# B&R Automation Studio project OpcUaSample410_BrbLibUa103 (part 15)

#### autoGeneratedFile.c - Auto generated code - list of all test sets in the program
```c
/*
B+R UnitTest: This is generated code.
Do not edit! Do not move!
Description: UnitTest Testprogramm infrastructure (List of TestSets).
LastUpdated: 2023-04-20 12:30:26Z
By B+R UnitTest Helper Version: 2.0.1.59
*/
#include "UnitTest.h"

UNITTEST_TESTSET_DECLARATION  Set_BrbUaClearVariantValue;
UNITTEST_TESTSET_DECLARATION  Set_BrbUaConvVariantValueFromString;
UNITTEST_TESTSET_DECLARATION  Set_BrbUaConvVariantValueToString;
UNITTEST_TESTSET_DECLARATION  Set_BrbUaAddVariantValueSubName;

UNITTEST_TESTSET_FIXTURES(utTestSets)
{
	new_TestSet(Set_BrbUaClearVariantValue),
	new_TestSet(Set_BrbUaConvVariantValueFromString),
	new_TestSet(Set_BrbUaConvVariantValueToString),
	new_TestSet(Set_BrbUaAddVariantValueSubName),
};
UNTITTEST_TESTSET_HANDLER();
```

#### Set_BrbUaClearVariantValue.c - Test set
```c
#include <bur/plctypes.h>

#ifdef _DEFAULT_INCLUDES
#include <AsDefault.h>
#endif

#include "UnitTest.h"
#include "BrbAsserts.h"
#include <string.h>

// NOLINTBEGIN(readability-*, bugprone-easily-swappable-parameters, bugprone-branch-clone, clang-diagnostic-invalid-utf8, clang-diagnostic-invalid-source-encoding, clang-diagnostic-pointer-arith, clang-diagnostic-strict-prototypes, clang-diagnostic-bad-function-cast, clang-analyzer-security.insecureAPI.*, hicpp-uppercase-literal-suffix, cppcoreguidelines-*, performance-*)
_TEST BrbUaClearVariantValue_NulPtr(void)
{
	dwordOut = BrbUaClearVariantValue(0);
	TEST_ASSERT_EQUAL_INT(0x80460000, dwordOut); // = Bad_StructureMissing

	// Finished
	TEST_DONE;
}

_TEST BrbUaClearVariantValue_Clear(void)
{
	memset(&variantIn0, 1, sizeof(variantIn0));
	variantIn0.VariantType = UAVariantType_Byte;
	dwordOut = BrbUaClearVariantValue(&variantIn0);
	TEST_ASSERT_EQUAL_INT(0x00000000, dwordOut); // = Good
	BRB_ASSERT_EQUAL_DINT(UAVariantType_Byte, (DINT)variantIn0.VariantType);

	// Finished
	TEST_DONE;
}

// NOLINTEND(readability-*, bugprone-easily-swappable-parameters, bugprone-branch-clone, clang-diagnostic-invalid-utf8, clang-diagnostic-invalid-source-encoding, clang-diagnostic-pointer-arith, clang-diagnostic-strict-prototypes, clang-diagnostic-bad-function-cast, clang-analyzer-security.insecureAPI.*, hicpp-uppercase-literal-suffix, cppcoreguidelines-*, performance-*)

/*
B+R UnitTest: This is generated code.
Do not edit! Do not move!
Description: UnitTest Testprogramm infrastructure (TestSet).
LastUpdated: 2023-04-20 10:55:13Z
By B+R UnitTest Helper Version: 2.0.1.59
*/
UNITTEST_FIXTURES(fixtures)
{
	new_TestFixture("BrbUaClearVariantValue_NulPtr", BrbUaClearVariantValue_NulPtr),
	new_TestFixture("BrbUaClearVariantValue_Clear", BrbUaClearVariantValue_Clear),
};

UNITTEST_CALLER_COMPLETE_EXPLICIT(Set_BrbUaClearVariantValue, "Set_BrbUaClearVariantValue", 0, 0, fixtures, 0, 0, 0);
```

#### Set_BrbUaConvVariantValueFromString.c - Test set
```c
#include <bur/plctypes.h>

#ifdef _DEFAULT_INCLUDES
#include <AsDefault.h>
#endif

#include "UnitTest.h"
#include "BrbAsserts.h"
#include <string.h>

// NOLINTBEGIN(readability-*, bugprone-easily-swappable-parameters, bugprone-branch-clone, clang-diagnostic-invalid-utf8, clang-diagnostic-invalid-source-encoding, clang-diagnostic-pointer-arith, clang-diagnostic-strict-prototypes, clang-diagnostic-bad-function-cast, clang-analyzer-security.insecureAPI.*, hicpp-uppercase-literal-suffix, cppcoreguidelines-*, performance-*)
_TEST BrbUaConvVariantValueFromString_NulPtr(void)
{
	dwordOut = BrbUaConvVariantValueFromString(0, stringIn0);
	TEST_ASSERT_EQUAL_INT(0x80460000, dwordOut); // = Bad_StructureMissing

	dwordOut = BrbUaConvVariantValueFromString(&variantIn0, 0);
	TEST_ASSERT_EQUAL_INT(0x80460000, dwordOut); // = Bad_StructureMissing

	// Finished
	TEST_DONE;
}

_TEST BrbUaConvVariantValueFromString_Boolean(void)
{
	memset(&variantIn0, 0, sizeof(variantIn0));
	variantIn0.VariantType = UAVariantType_Boolean;
	strcpy(stringIn0, "xxx");
	dwordOut = BrbUaConvVariantValueFromString(&variantIn0, stringIn0);
	TEST_ASSERT_EQUAL_INT(0x00000000, dwordOut); // = Good
	BRB_ASSERT_EQUAL_DINT(UAVariantType_Boolean, (DINT)variantIn0.VariantType);
	BRB_ASSERT_EQUAL_BOOL(0, variantIn0.Boolean);

	memset(&variantIn0, 0, sizeof(variantIn0));
	variantIn0.VariantType = UAVariantType_Boolean;
	strcpy(stringIn0, "0");
	dwordOut = BrbUaConvVariantValueFromString(&variantIn0, stringIn0);
	TEST_ASSERT_EQUAL_INT(0x00000000, dwordOut); // = Good
	BRB_ASSERT_EQUAL_DINT(UAVariantType_Boolean, (DINT)variantIn0.VariantType);
	BRB_ASSERT_EQUAL_BOOL(0, variantIn0.Boolean);

	memset(&variantIn0, 0, sizeof(variantIn0));
	variantIn0.VariantType = UAVariantType_Boolean;
	strcpy(stringIn0, "False");
	dwordOut = BrbUaConvVariantValueFromString(&variantIn0, stringIn0);
	TEST_ASSERT_EQUAL_INT(0x00000000, dwordOut); // = Good
	BRB_ASSERT_EQUAL_DINT(UAVariantType_Boolean, (DINT)variantIn0.VariantType);
	BRB_ASSERT_EQUAL_BOOL(0, variantIn0.Boolean);

	memset(&variantIn0, 0, sizeof(variantIn0));
	variantIn0.VariantType = UAVariantType_Boolean;
	strcpy(stringIn0, "false");
	dwordOut = BrbUaConvVariantValueFromString(&variantIn0, stringIn0);
	TEST_ASSERT_EQUAL_INT(0x00000000, dwordOut); // = Good
	BRB_ASSERT_EQUAL_DINT(UAVariantType_Boolean, (DINT)variantIn0.VariantType);
	BRB_ASSERT_EQUAL_BOOL(0, variantIn0.Boolean);

	memset(&variantIn0, 0, sizeof(variantIn0));
	variantIn0.VariantType = UAVariantType_Boolean;
	strcpy(stringIn0, "1");
	dwordOut = BrbUaConvVariantValueFromString(&variantIn0, stringIn0);
	TEST_ASSERT_EQUAL_INT(0x00000000, dwordOut); // = Good
	BRB_ASSERT_EQUAL_DINT(UAVariantType_Boolean, (DINT)variantIn0.VariantType);
	BRB_ASSERT_EQUAL_BOOL(1, variantIn0.Boolean);

	memset(&variantIn0, 0, sizeof(variantIn0));
	variantIn0.VariantType = UAVariantType_Boolean;
	strcpy(stringIn0, "True");
	dwordOut = BrbUaConvVariantValueFromString(&variantIn0, stringIn0);
	TEST_ASSERT_EQUAL_INT(0x00000000, dwordOut); // = Good
	BRB_ASSERT_EQUAL_DINT(UAVariantType_Boolean, (DINT)variantIn0.VariantType);
	BRB_ASSERT_EQUAL_BOOL(1, variantIn0.Boolean);

	memset(&variantIn0, 0, sizeof(variantIn0));
	variantIn0.VariantType = UAVariantType_Boolean;
	strcpy(stringIn0, "true");
	dwordOut = BrbUaConvVariantValueFromString(&variantIn0, stringIn0);
	TEST_ASSERT_EQUAL_INT(0x00000000, dwordOut); // = Good
	BRB_ASSERT_EQUAL_DINT(UAVariantType_Boolean, (DINT)variantIn0.VariantType);
	BRB_ASSERT_EQUAL_BOOL(1, variantIn0.Boolean);

	// Finished
	TEST_DONE;
}

_TEST BrbUaConvVariantValueFromString_SByte(void)
{
	memset(&variantIn0, 0, sizeof(variantIn0));
	variantIn0.VariantType = UAVariantType_SByte;
	strcpy(stringIn0, "-128");
	dwordOut = BrbUaConvVariantValueFromString(&variantIn0, stringIn0);
	TEST_ASSERT_EQUAL_INT(0x00000000, dwordOut); // = Good
	BRB_ASSERT_EQUAL_DINT(UAVariantType_SByte, (DINT)variantIn0.VariantType);
	BRB_ASSERT_EQUAL_DINT(-128, (DINT)variantIn0.SByte);

	// Finished
	TEST_DONE;
}

_TEST BrbUaConvVariantValueFromString_Byte(void)
{
	memset(&variantIn0, 0, sizeof(variantIn0));
	variantIn0.VariantType = UAVariantType_Byte;
	strcpy(stringIn0, "127");
	dwordOut = BrbUaConvVariantValueFromString(&variantIn0, stringIn0);
	TEST_ASSERT_EQUAL_INT(0x00000000, dwordOut); // = Good
	BRB_ASSERT_EQUAL_DINT(UAVariantType_Byte, (DINT)variantIn0.VariantType);
	BRB_ASSERT_EQUAL_UDINT(127, (UDINT)variantIn0.Byte);

	// Finished
	TEST_DONE;
}

_TEST BrbUaConvVariantValueFromString_Int16(void)
{
	memset(&variantIn0, 0, sizeof(variantIn0));
	variantIn0.VariantType = UAVariantType_Int16;
	strcpy(stringIn0, "-32768");
	dwordOut = BrbUaConvVariantValueFromString(&variantIn0, stringIn0);
	TEST_ASSERT_EQUAL_INT(0x00000000, dwordOut); // = Good
	BRB_ASSERT_EQUAL_DINT(UAVariantType_Int16, (DINT)variantIn0.VariantType);
	BRB_ASSERT_EQUAL_DINT(-32768, (DINT)variantIn0.Int16);

	// Finished
	TEST_DONE;
}

_TEST BrbUaConvVariantValueFromString_Uint16(void)
{
	memset(&variantIn0, 0, sizeof(variantIn0));
	variantIn0.VariantType = UAVariantType_UInt16;
	strcpy(stringIn0, "65535");
	dwordOut = BrbUaConvVariantValueFromString(&variantIn0, stringIn0);
	TEST_ASSERT_EQUAL_INT(0x00000000, dwordOut); // = Good
	BRB_ASSERT_EQUAL_DINT(UAVariantType_UInt16, (DINT)variantIn0.VariantType);
	BRB_ASSERT_EQUAL_UDINT(65535, (UDINT)variantIn0.UInt16);

	// Finished
	TEST_DONE;
}

_TEST BrbUaConvVariantValueFromString_Int32(void)
{
	memset(&variantIn0, 0, sizeof(variantIn0));
	variantIn0.VariantType = UAVariantType_Int32;
	strcpy(stringIn0, "-2147483648");
	dwordOut = BrbUaConvVariantValueFromString(&variantIn0, stringIn0);
	TEST_ASSERT_EQUAL_INT(0x00000000, dwordOut); // = Good
	BRB_ASSERT_EQUAL_DINT(UAVariantType_Int32, (DINT)variantIn0.VariantType);
	BRB_ASSERT_EQUAL_DINT(-2147483648, (DINT)variantIn0.Int32);

	// Finished
	TEST_DONE;
}

_TEST BrbUaConvVariantValueFromString_Uint32(void)
{
	memset(&variantIn0, 0, sizeof(variantIn0));
	variantIn0.VariantType = UAVariantType_UInt32;
	strcpy(stringIn0, "4294967295");
	dwordOut = BrbUaConvVariantValueFromString(&variantIn0, stringIn0);
	TEST_ASSERT_EQUAL_INT(0x00000000, dwordOut); // = Good
	BRB_ASSERT_EQUAL_DINT(UAVariantType_UInt32, (DINT)variantIn0.VariantType);
	BRB_ASSERT_EQUAL_UDINT(4294967295, variantIn0.UInt32);

	// Finished
	TEST_DONE;
}

_TEST BrbUaConvVariantValueFromString_Int64(void)
{
	memset(&variantIn0, 0, sizeof(variantIn0));
	variantIn0.VariantType = UAVariantType_Int64;
	strcpy(stringIn0, "-2147483648");
	dwordOut = BrbUaConvVariantValueFromString(&variantIn0, stringIn0);
	TEST_ASSERT_EQUAL_INT(0x803D0000, dwordOut); // = Bad_NotSupported
	BRB_ASSERT_EQUAL_DINT(UAVariantType_Int64, (DINT)variantIn0.VariantType);

	// Finished
	TEST_DONE;
}

_TEST BrbUaConvVariantValueFromString_Uint64(void)
{
	memset(&variantIn0, 0, sizeof(variantIn0));
	variantIn0.VariantType = UAVariantType_UInt64;
	strcpy(stringIn0, "4294967295");
	dwordOut = BrbUaConvVariantValueFromString(&variantIn0, stringIn0);
	TEST_ASSERT_EQUAL_INT(0x803D0000, dwordOut); // = Bad_NotSupported
	BRB_ASSERT_EQUAL_DINT(UAVariantType_UInt64, (DINT)variantIn0.VariantType);

	// Finished
	TEST_DONE;
}

_TEST BrbUaConvVariantValueFromString_Float(void)
{
	memset(&variantIn0, 0, sizeof(variantIn0));
	variantIn0.VariantType = UAVariantType_Float;
	strcpy(stringIn0, "-1.23");
	dwordOut = BrbUaConvVariantValueFromString(&variantIn0, stringIn0);
	TEST_ASSERT_EQUAL_INT(0x00000000, dwordOut); // = Good
	BRB_ASSERT_EQUAL_DINT(UAVariantType_Float, (DINT)variantIn0.VariantType);
	TEST_ASSERT_EQUAL_REAL(-1.23, variantIn0.Float);

	// Finished
	TEST_DONE;
}

_TEST BrbUaConvVariantValueFromString_Double(void)
{
	memset(&variantIn0, 0, sizeof(variantIn0));
	variantIn0.VariantType = UAVariantType_Double;
	strcpy(stringIn0, "-2.34");
	dwordOut = BrbUaConvVariantValueFromString(&variantIn0, stringIn0);
	TEST_ASSERT_EQUAL_INT(0x00000000, dwordOut); // = Good
	BRB_ASSERT_EQUAL_DINT(UAVariantType_Double, (DINT)variantIn0.VariantType);
	TEST_ASSERT_EQUAL_LREAL((LREAL)-2.3399999141693115, variantIn0.Double);

	// Finished
	TEST_DONE;
}

_TEST BrbUaConvVariantValueFromString_String(void)
{
	memset(&variantIn0, 0, sizeof(variantIn0));
	variantIn0.VariantType = UAVariantType_String;
	strcpy(stringIn0, "Hallo");
	dwordOut = BrbUaConvVariantValueFromString(&variantIn0, stringIn0);
	TEST_ASSERT_EQUAL_INT(0x00000000, dwordOut); // = Good
	BRB_ASSERT_EQUAL_DINT(UAVariantType_String, (DINT)variantIn0.VariantType);
	TEST_ASSERT_EQUAL_STRING("Hallo", variantIn0.String);

	// Finished
	TEST_DONE;
}

_TEST BrbUaConvVariantValueFromString_DateTime(void)
{
	memset(&variantIn0, 0, sizeof(variantIn0));
	variantIn0.VariantType = UAVariantType_DateTime;
	strcpy(stringIn0, "2106.02.07 06:28:15:000:000");
	dwordOut = BrbUaConvVariantValueFromString(&variantIn0, stringIn0);
	TEST_ASSERT_EQUAL_INT(0x00000000, dwordOut); // = Good
	BRB_ASSERT_EQUAL_DINT(UAVariantType_DateTime, (DINT)variantIn0.VariantType);
	BRB_ASSERT_EQUAL_UDINT(4294967295, (UDINT)variantIn0.DateTime);

	// Finished
	TEST_DONE;
}

_TEST BrbUaConvVariantValueFromString_Guid(void)
{
	memset(&variantIn0, 0, sizeof(variantIn0));
	variantIn0.VariantType = UAVariantType_Guid;
	strcpy(stringIn0, "12345678-1234-5678-9ABC-123456789ABC");
	dwordOut = BrbUaConvVariantValueFromString(&variantIn0, stringIn0);
	TEST_ASSERT_EQUAL_INT(0x00000000, dwordOut); // = Good
	BRB_ASSERT_EQUAL_DINT(UAVariantType_Guid, (DINT)variantIn0.VariantType);
	TEST_ASSERT_EQUAL_STRING("12345678-1234-5678-9ABC-123456789ABC", variantIn0.String);

	// Finished
	TEST_DONE;
}

_TEST BrbUaConvVariantValueFromString_ByteString(void)
{
	memset(&variantIn0, 0, sizeof(variantIn0));
	variantIn0.VariantType = UAVariantType_ByteString;
	strcpy(stringIn0, "123456789ABC");
	dwordOut = BrbUaConvVariantValueFromString(&variantIn0, stringIn0);
	TEST_ASSERT_EQUAL_INT(0x803D0000, dwordOut); // = Bad_NotSupported
	BRB_ASSERT_EQUAL_DINT(UAVariantType_ByteString, (DINT)variantIn0.VariantType);

	// Finished
	TEST_DONE;
}

_TEST BrbUaConvVariantValueFromString_XmlElement(void)
{
	memset(&variantIn0, 0, sizeof(variantIn0));
	variantIn0.VariantType = UAVariantType_XmlElement;
	strcpy(stringIn0, "<Hallo >");
	dwordOut = BrbUaConvVariantValueFromString(&variantIn0, stringIn0);
	TEST_ASSERT_EQUAL_INT(0x803D0000, dwordOut); // = Bad_NotSupported
	BRB_ASSERT_EQUAL_DINT(UAVariantType_XmlElement, (DINT)variantIn0.VariantType);

	// Finished
	TEST_DONE;
}

_TEST BrbUaConvVariantValueFromString_NodeId(void)
{
	memset(&variantIn0, 0, sizeof(variantIn0));
	variantIn0.VariantType = UAVariantType_NodeId;
	strcpy(stringIn0, "ns=34");
	dwordOut = BrbUaConvVariantValueFromString(&variantIn0, stringIn0);
	TEST_ASSERT_EQUAL_INT(0x80330000 , dwordOut); // = Bad_NodeIdInvalid
	BRB_ASSERT_EQUAL_DINT(UAVariantType_NodeId, (DINT)variantIn0.VariantType);
	BRB_ASSERT_EQUAL_UDINT(34, (UDINT)variantIn0.NodeId.NamespaceIndex);
	//BRB_ASSERT_EQUAL_DINT(UAIdentifierType_Numeric, variantIn0.NodeId.IdentifierType);
	TEST_ASSERT_EQUAL_STRING("", variantIn0.NodeId.Identifier);

	memset(&variantIn0, 0, sizeof(variantIn0));
	variantIn0.VariantType = UAVariantType_NodeId;
	strcpy(stringIn0, "ns=56;");
	dwordOut = BrbUaConvVariantValueFromString(&variantIn0, stringIn0);
	TEST_ASSERT_EQUAL_INT(0x80330000 , dwordOut); // = Bad_NodeIdInvalid
	BRB_ASSERT_EQUAL_DINT(UAVariantType_NodeId, (DINT)variantIn0.VariantType);
	BRB_ASSERT_EQUAL_UDINT(56, (UDINT)variantIn0.NodeId.NamespaceIndex);
	//BRB_ASSERT_EQUAL_DINT(UAIdentifierType_Numeric, variantIn0.NodeId.IdentifierType);
	TEST_ASSERT_EQUAL_STRING("", variantIn0.NodeId.Identifier);

	memset(&variantIn0, 0, sizeof(variantIn0));
	variantIn0.VariantType = UAVariantType_NodeId;
	strcpy(stringIn0, "ns=123;v=Hallo");
	dwordOut = BrbUaConvVariantValueFromString(&variantIn0, stringIn0);
	TEST_ASSERT_EQUAL_INT(0x80330000 , dwordOut); // = Bad_NodeIdInvalid
	BRB_ASSERT_EQUAL_DINT(UAVariantType_NodeId, (DINT)variantIn0.VariantType);
	BRB_ASSERT_EQUAL_UDINT(123, (UDINT)variantIn0.NodeId.NamespaceIndex);
	//BRB_ASSERT_EQUAL_DINT(UAIdentifierType_Numeric, variantIn0.NodeId.IdentifierType);
	TEST_ASSERT_EQUAL_STRING("", variantIn0.NodeId.Identifier);

	memset(&variantIn0, 0, sizeof(variantIn0));
	variantIn0.VariantType = UAVariantType_NodeId;
	strcpy(stringIn0, "i=1234");
	dwordOut = BrbUaConvVariantValueFromString(&variantIn0, stringIn0);
	TEST_ASSERT_EQUAL_INT(0x00000000, dwordOut); // = Good
	BRB_ASSERT_EQUAL_DINT(UAVariantType_NodeId, (DINT)variantIn0.VariantType);
	BRB_ASSERT_EQUAL_UDINT(0, (UDINT)variantIn0.NodeId.NamespaceIndex);
	BRB_ASSERT_EQUAL_DINT(UAIdentifierType_Numeric, (DINT)variantIn0.NodeId.IdentifierType);
	TEST_ASSERT_EQUAL_STRING("1234", variantIn0.NodeId.Identifier);

	memset(&variantIn0, 0, sizeof(variantIn0));
	variantIn0.VariantType = UAVariantType_NodeId;
	strcpy(stringIn0, "ns=21;i=2345");
	dwordOut = BrbUaConvVariantValueFromString(&variantIn0, stringIn0);
	TEST_ASSERT_EQUAL_INT(0x00000000, dwordOut); // = Good
	BRB_ASSERT_EQUAL_DINT(UAVariantType_NodeId, (DINT)variantIn0.VariantType);
	BRB_ASSERT_EQUAL_UDINT(21, (UDINT)variantIn0.NodeId.NamespaceIndex);
	BRB_ASSERT_EQUAL_DINT(UAIdentifierType_Numeric, (DINT)variantIn0.NodeId.IdentifierType);
	TEST_ASSERT_EQUAL_STRING("2345", variantIn0.NodeId.Identifier);

	memset(&variantIn0, 0, sizeof(variantIn0));
	variantIn0.VariantType = UAVariantType_NodeId;
	strcpy(stringIn0, "s=Hallo");
	dwordOut = BrbUaConvVariantValueFromString(&variantIn0, stringIn0);
	TEST_ASSERT_EQUAL_INT(0x00000000, dwordOut); // = Good
	BRB_ASSERT_EQUAL_DINT(UAVariantType_NodeId, (DINT)variantIn0.VariantType);
	BRB_ASSERT_EQUAL_UDINT(0, (UDINT)variantIn0.NodeId.NamespaceIndex);
	BRB_ASSERT_EQUAL_DINT(UAIdentifierType_String, (DINT)variantIn0.NodeId.IdentifierType);
	TEST_ASSERT_EQUAL_STRING("Hallo", variantIn0.NodeId.Identifier);

	memset(&variantIn0, 0, sizeof(variantIn0));
	variantIn0.VariantType = UAVariantType_NodeId;
	strcpy(stringIn0, "ns=22;s=Hello");
	dwordOut = BrbUaConvVariantValueFromString(&variantIn0, stringIn0);
	TEST_ASSERT_EQUAL_INT(0x00000000, dwordOut); // = Good
	BRB_ASSERT_EQUAL_DINT(UAVariantType_NodeId, (DINT)variantIn0.VariantType);
	BRB_ASSERT_EQUAL_UDINT(22, (UDINT)variantIn0.NodeId.NamespaceIndex);
	BRB_ASSERT_EQUAL_DINT(UAIdentifierType_String, (DINT)variantIn0.NodeId.IdentifierType);
	TEST_ASSERT_EQUAL_STRING("Hello", variantIn0.NodeId.Identifier);

	memset(&variantIn0, 0, sizeof(variantIn0));
	variantIn0.VariantType = UAVariantType_NodeId;
	strcpy(stringIn0, "g=7fdf25f9-7815-e783-488b-a4247f55b88e");
	dwordOut = BrbUaConvVariantValueFromString(&variantIn0, stringIn0);
	TEST_ASSERT_EQUAL_INT(0x00000000, dwordOut); // = Good
	BRB_ASSERT_EQUAL_DINT(UAVariantType_NodeId, (DINT)variantIn0.VariantType);
	BRB_ASSERT_EQUAL_UDINT(0, (UDINT)variantIn0.NodeId.NamespaceIndex);
	BRB_ASSERT_EQUAL_DINT(UAIdentifierType_GUID, (DINT)variantIn0.NodeId.IdentifierType);
	TEST_ASSERT_EQUAL_STRING("7fdf25f9-7815-e783-488b-a4247f55b88e", variantIn0.NodeId.Identifier);

	memset(&variantIn0, 0, sizeof(variantIn0));
	variantIn0.VariantType = UAVariantType_NodeId;
	strcpy(stringIn0, "ns=23;g=80e0360a-7815-e783-488b-a4247f55b88e");
	dwordOut = BrbUaConvVariantValueFromString(&variantIn0, stringIn0);
	TEST_ASSERT_EQUAL_INT(0x00000000, dwordOut); // = Good
	BRB_ASSERT_EQUAL_DINT(UAVariantType_NodeId, (DINT)variantIn0.VariantType);
	BRB_ASSERT_EQUAL_UDINT(23, (UDINT)variantIn0.NodeId.NamespaceIndex);
	BRB_ASSERT_EQUAL_DINT(UAIdentifierType_GUID, (DINT)variantIn0.NodeId.IdentifierType);
	TEST_ASSERT_EQUAL_STRING("80e0360a-7815-e783-488b-a4247f55b88e", variantIn0.NodeId.Identifier);

	// Finished
	TEST_DONE;
}

_TEST BrbUaConvVariantValueFromString_ExpandedNodeId(void)
{
	memset(&variantIn0, 0, sizeof(variantIn0));
	variantIn0.VariantType = UAVariantType_ExpandedNodeId;
	strcpy(stringIn0, "xxxyyy");
	dwordOut = BrbUaConvVariantValueFromString(&variantIn0, stringIn0);
	TEST_ASSERT_EQUAL_INT(0x803D0000, dwordOut); // = Bad_NotSupported
	BRB_ASSERT_EQUAL_DINT(UAVariantType_ExpandedNodeId, (DINT)variantIn0.VariantType);

	// Finished
	TEST_DONE;
}

_TEST BrbUaConvVariantValueFromString_StatusCode(void)
{
	memset(&variantIn0, 0, sizeof(variantIn0));
	variantIn0.VariantType = UAVariantType_StatusCode;
	strcpy(stringIn0, "32987");
	dwordOut = BrbUaConvVariantValueFromString(&variantIn0, stringIn0);
	TEST_ASSERT_EQUAL_INT(0x00000000, dwordOut); // = Good
	BRB_ASSERT_EQUAL_DINT(UAVariantType_StatusCode, (DINT)variantIn0.VariantType);
	BRB_ASSERT_EQUAL_UDINT(32987, variantIn0.UInt32);

	memset(&variantIn0, 0, sizeof(variantIn0));
	variantIn0.VariantType = UAVariantType_StatusCode;
	strcpy(stringIn0, "0xA0150000");
	dwordOut = BrbUaConvVariantValueFromString(&variantIn0, stringIn0);
	TEST_ASSERT_EQUAL_INT(0x00000000, dwordOut); // = Good
	BRB_ASSERT_EQUAL_DINT(UAVariantType_StatusCode, (DINT)variantIn0.VariantType);
	BRB_ASSERT_EQUAL_UDINT(2685730816, variantIn0.UInt32);

	// Finished
	TEST_DONE;
}

_TEST BrbUaConvVariantValueFromString_QualifiedName(void)
{
	memset(&variantIn0, 0, sizeof(variantIn0));
	variantIn0.VariantType = UAVariantType_QualifiedName;
	strcpy(stringIn0, "xxxyyy");
	dwordOut = BrbUaConvVariantValueFromString(&variantIn0, stringIn0);
	TEST_ASSERT_EQUAL_INT(0x803D0000, dwordOut); // = Bad_NotSupported
	BRB_ASSERT_EQUAL_DINT(UAVariantType_QualifiedName, (DINT)variantIn0.VariantType);

	// Finished
	TEST_DONE;
}

_TEST BrbUaConvVariantValueFromString_LocalizedText(void)
{
	memset(&variantIn0, 0, sizeof(variantIn0));
	variantIn0.VariantType = UAVariantType_LocalizedText;
	strcpy(stringIn0, "xxxyyy");
	dwordOut = BrbUaConvVariantValueFromString(&variantIn0, stringIn0);
	TEST_ASSERT_EQUAL_INT(0x803D0000, dwordOut); // = Bad_NotSupported
	BRB_ASSERT_EQUAL_DINT(UAVariantType_LocalizedText, (DINT)variantIn0.VariantType);

	// Finished
	TEST_DONE;
}

// NOLINTEND(readability-*, bugprone-easily-swappable-parameters, bugprone-branch-clone, clang-diagnostic-invalid-utf8, clang-diagnostic-invalid-source-encoding, clang-diagnostic-pointer-arith, clang-diagnostic-strict-prototypes, clang-diagnostic-bad-function-cast, clang-analyzer-security.insecureAPI.*, hicpp-uppercase-literal-suffix, cppcoreguidelines-*, performance-*)

/*
B+R UnitTest: This is generated code.
Do not edit! Do not move!
Description: UnitTest Testprogramm infrastructure (TestSet).
LastUpdated: 2023-05-04 13:01:25Z
By B+R UnitTest Helper Version: 2.0.1.59
*/
UNITTEST_FIXTURES(fixtures)
{
	new_TestFixture("BrbUaConvVariantValueFromString_NulPtr", BrbUaConvVariantValueFromString_NulPtr),
	new_TestFixture("BrbUaConvVariantValueFromString_Boolean", BrbUaConvVariantValueFromString_Boolean),
	new_TestFixture("BrbUaConvVariantValueFromString_SByte", BrbUaConvVariantValueFromString_SByte),
	new_TestFixture("BrbUaConvVariantValueFromString_Byte", BrbUaConvVariantValueFromString_Byte),
	new_TestFixture("BrbUaConvVariantValueFromString_Int16", BrbUaConvVariantValueFromString_Int16),
	new_TestFixture("BrbUaConvVariantValueFromString_Uint16", BrbUaConvVariantValueFromString_Uint16),
	new_TestFixture("BrbUaConvVariantValueFromString_Int32", BrbUaConvVariantValueFromString_Int32),
	new_TestFixture("BrbUaConvVariantValueFromString_Uint32", BrbUaConvVariantValueFromString_Uint32),
	new_TestFixture("BrbUaConvVariantValueFromString_Int64", BrbUaConvVariantValueFromString_Int64),
	new_TestFixture("BrbUaConvVariantValueFromString_Uint64", BrbUaConvVariantValueFromString_Uint64),
	new_TestFixture("BrbUaConvVariantValueFromString_Float", BrbUaConvVariantValueFromString_Float),
	new_TestFixture("BrbUaConvVariantValueFromString_Double", BrbUaConvVariantValueFromString_Double),
	new_TestFixture("BrbUaConvVariantValueFromString_String", BrbUaConvVariantValueFromString_String),
	new_TestFixture("BrbUaConvVariantValueFromString_DateTime", BrbUaConvVariantValueFromString_DateTime),
	new_TestFixture("BrbUaConvVariantValueFromString_Guid", BrbUaConvVariantValueFromString_Guid),
	new_TestFixture("BrbUaConvVariantValueFromString_ByteString", BrbUaConvVariantValueFromString_ByteString),
	new_TestFixture("BrbUaConvVariantValueFromString_XmlElement", BrbUaConvVariantValueFromString_XmlElement),
	new_TestFixture("BrbUaConvVariantValueFromString_NodeId", BrbUaConvVariantValueFromString_NodeId),
	new_TestFixture("BrbUaConvVariantValueFromString_ExpandedNodeId", BrbUaConvVariantValueFromString_ExpandedNodeId),
	new_TestFixture("BrbUaConvVariantValueFromString_StatusCode", BrbUaConvVariantValueFromString_StatusCode),
	new_TestFixture("BrbUaConvVariantValueFromString_QualifiedName", BrbUaConvVariantValueFromString_QualifiedName),
	new_TestFixture("BrbUaConvVariantValueFromString_LocalizedText", BrbUaConvVariantValueFromString_LocalizedText),
};

UNITTEST_CALLER_COMPLETE_EXPLICIT(Set_BrbUaConvVariantValueFromString, "Set_BrbUaConvVariantValueFromString", 0, 0, fixtures, 0, 0, 0);
```

#### Set_BrbUaConvVariantValueToString.c - Test set
```c
#include <bur/plctypes.h>

#ifdef _DEFAULT_INCLUDES
#include <AsDefault.h>
#endif

#include "UnitTest.h"
#include "BrbAsserts.h"
#include <string.h>

// NOLINTBEGIN(readability-*, bugprone-easily-swappable-parameters, bugprone-branch-clone, clang-diagnostic-invalid-utf8, clang-diagnostic-invalid-source-encoding, clang-diagnostic-pointer-arith, clang-diagnostic-strict-prototypes, clang-diagnostic-bad-function-cast, clang-analyzer-security.insecureAPI.*, hicpp-uppercase-literal-suffix, cppcoreguidelines-*, performance-*)
_TEST BrbUaConvVariantValueToString_NulPtr(void)
{
	dwordOut = BrbUaConvVariantValueToString(0, stringIn0, sizeof(stringIn0));
	TEST_ASSERT_EQUAL_INT(0x80460000, dwordOut); // = Bad_StructureMissing

	dwordOut = BrbUaConvVariantValueToString(&variantIn0, 0, sizeof(stringIn0));
	TEST_ASSERT_EQUAL_INT(0x80460000, dwordOut); // = Bad_StructureMissing

	// Finished
	TEST_DONE;
}

_TEST BrbUaConvVariantValueToString_Bool(void)
{
	memset(&variantIn0, 0, sizeof(variantIn0));
	variantIn0.VariantType = UAVariantType_Boolean;
	variantIn0.Boolean = 0;
	dwordOut = BrbUaConvVariantValueToString(&variantIn0, stringIn0, sizeof(stringIn0));
	TEST_ASSERT_EQUAL_INT(0x00000000, dwordOut); // = Good
	BRB_ASSERT_EQUAL_DINT(UAVariantType_Boolean, (DINT)variantIn0.VariantType);
	TEST_ASSERT_EQUAL_STRING("False", stringIn0);

	memset(&variantIn0, 0, sizeof(variantIn0));
	variantIn0.VariantType = UAVariantType_Boolean;
	variantIn0.Boolean = 1;
	dwordOut = BrbUaConvVariantValueToString(&variantIn0, stringIn0, sizeof(stringIn0));
	TEST_ASSERT_EQUAL_INT(0x00000000, dwordOut); // = Good
	BRB_ASSERT_EQUAL_DINT(UAVariantType_Boolean, (DINT)variantIn0.VariantType);
	TEST_ASSERT_EQUAL_STRING("True", stringIn0);

	// Finished
	TEST_DONE;
}

_TEST BrbUaConvVariantValueToString_SByte(void)
{
	memset(&variantIn0, 0, sizeof(variantIn0));
	variantIn0.VariantType = UAVariantType_SByte;
	variantIn0.SByte = -128;
	dwordOut = BrbUaConvVariantValueToString(&variantIn0, stringIn0, sizeof(stringIn0));
	TEST_ASSERT_EQUAL_INT(0x00000000, dwordOut); // = Good
	BRB_ASSERT_EQUAL_DINT(UAVariantType_SByte, (DINT)variantIn0.VariantType);
	TEST_ASSERT_EQUAL_STRING("-128", stringIn0);

	// Finished
	TEST_DONE;
}

_TEST BrbUaConvVariantValueToString_Byte(void)
{
	memset(&variantIn0, 0, sizeof(variantIn0));

	variantIn0.VariantType = UAVariantType_Byte;
	variantIn0.Byte = 255;
	dwordOut = BrbUaConvVariantValueToString(&variantIn0, stringIn0, sizeof(stringIn0));
	TEST_ASSERT_EQUAL_INT(0x00000000, dwordOut); // = Good
	BRB_ASSERT_EQUAL_DINT(UAVariantType_Byte, (DINT)variantIn0.VariantType);
	TEST_ASSERT_EQUAL_STRING("255", stringIn0);

	// Finished
	TEST_DONE;
}

_TEST BrbUaConvVariantValueToString_Int16(void)
{
	memset(&variantIn0, 0, sizeof(variantIn0));
	variantIn0.VariantType = UAVariantType_Int16;
	variantIn0.Int16 = -32768;
	dwordOut = BrbUaConvVariantValueToString(&variantIn0, stringIn0, sizeof(stringIn0));
	TEST_ASSERT_EQUAL_INT(0x00000000, dwordOut); // = Good
	BRB_ASSERT_EQUAL_DINT(UAVariantType_Int16, (DINT)variantIn0.VariantType);
	TEST_ASSERT_EQUAL_STRING("-32768", stringIn0);

	// Finished
	TEST_DONE;
}

_TEST BrbUaConvVariantValueToString_UInt16(void)
{
	memset(&variantIn0, 0, sizeof(variantIn0));
	variantIn0.VariantType = UAVariantType_UInt16;
	variantIn0.UInt16 = 65535;
	dwordOut = BrbUaConvVariantValueToString(&variantIn0, stringIn0, sizeof(stringIn0));
	TEST_ASSERT_EQUAL_INT(0x00000000, dwordOut); // = Good
	BRB_ASSERT_EQUAL_DINT(UAVariantType_UInt16, (DINT)variantIn0.VariantType);
	TEST_ASSERT_EQUAL_STRING("65535", stringIn0);

	// Finished
	TEST_DONE;
}

_TEST BrbUaConvVariantValueToString_Int32(void)
{
	memset(&variantIn0, 0, sizeof(variantIn0));
	variantIn0.VariantType = UAVariantType_Int32;
	variantIn0.Int32 = -2147483648;
	dwordOut = BrbUaConvVariantValueToString(&variantIn0, stringIn0, sizeof(stringIn0));
	TEST_ASSERT_EQUAL_INT(0x00000000, dwordOut); // = Good
	BRB_ASSERT_EQUAL_DINT(UAVariantType_Int32, (DINT)variantIn0.VariantType);
	TEST_ASSERT_EQUAL_STRING("-2147483648", stringIn0);

	// Finished
	TEST_DONE;
}

_TEST BrbUaConvVariantValueToString_UInt32(void)
{
	memset(&variantIn0, 0, sizeof(variantIn0));
	variantIn0.VariantType = UAVariantType_UInt32;
	strcpy(stringIn0, "4294967295");
	variantIn0.UInt32 = 4294967295;
	dwordOut = BrbUaConvVariantValueToString(&variantIn0, stringIn0, sizeof(stringIn0));
	TEST_ASSERT_EQUAL_INT(0x00000000, dwordOut); // = Good
	BRB_ASSERT_EQUAL_DINT(UAVariantType_UInt32, (DINT)variantIn0.VariantType);
	TEST_ASSERT_EQUAL_STRING("4294967295", stringIn0);

	// Finished
	TEST_DONE;
}

_TEST BrbUaConvVariantValueToString_Int64(void)
{
	memset(&variantIn0, 0, sizeof(variantIn0));
	variantIn0.VariantType = UAVariantType_Int64;
	dwordOut = BrbUaConvVariantValueToString(&variantIn0, stringIn0, sizeof(stringIn0));
	TEST_ASSERT_EQUAL_INT(0x803D0000, dwordOut); // = Bad_NotSupported
	BRB_ASSERT_EQUAL_DINT(UAVariantType_Int64, (DINT)variantIn0.VariantType);

	// Finished
	TEST_DONE;
}

_TEST BrbUaConvVariantValueToString_UInt64(void)
{
	memset(&variantIn0, 0, sizeof(variantIn0));
	variantIn0.VariantType = UAVariantType_UInt64;
	dwordOut = BrbUaConvVariantValueToString(&variantIn0, stringIn0, sizeof(stringIn0));
	TEST_ASSERT_EQUAL_INT(0x803D0000, dwordOut); // = Bad_NotSupported
	BRB_ASSERT_EQUAL_DINT(UAVariantType_UInt64, (DINT)variantIn0.VariantType);

	// Finished
	TEST_DONE;
}

_TEST BrbUaConvVariantValueToString_Float(void)
{
	memset(&variantIn0, 0, sizeof(variantIn0));
	variantIn0.VariantType = UAVariantType_Float;
	variantIn0.Float = -1.23f;
	dwordOut = BrbUaConvVariantValueToString(&variantIn0, stringIn0, sizeof(stringIn0));
	TEST_ASSERT_EQUAL_INT(0x00000000, dwordOut); // = Good
	BRB_ASSERT_EQUAL_DINT(UAVariantType_Float, (DINT)variantIn0.VariantType);
	TEST_ASSERT_EQUAL_STRING("-1.23", stringIn0);

	// Finished
	TEST_DONE;
}

_TEST BrbUaConvVariantValueToString_Double(void)
{
	memset(&variantIn0, 0, sizeof(variantIn0));
	variantIn0.VariantType = UAVariantType_Double;
	variantIn0.Double = (LREAL)-2.34;
	dwordOut = BrbUaConvVariantValueToString(&variantIn0, stringIn0, sizeof(stringIn0));
	TEST_ASSERT_EQUAL_INT(0x00000000, dwordOut); // = Good
	BRB_ASSERT_EQUAL_DINT(UAVariantType_Double, (DINT)variantIn0.VariantType);
	TEST_ASSERT_EQUAL_STRING("-2.34", stringIn0);

	// Finished
	TEST_DONE;
}

_TEST BrbUaConvVariantValueToString_String(void)
{
	memset(&variantIn0, 0, sizeof(variantIn0));
	variantIn0.VariantType = UAVariantType_String;
	strcpy(variantIn0.String, "Hallo");
	dwordOut = BrbUaConvVariantValueToString(&variantIn0, stringIn0, sizeof(stringIn0));
	TEST_ASSERT_EQUAL_INT(0x00000000, dwordOut); // = Good
	BRB_ASSERT_EQUAL_DINT(UAVariantType_String, (DINT)variantIn0.VariantType);
	TEST_ASSERT_EQUAL_STRING("Hallo", stringIn0);

	// Finished
	TEST_DONE;
}

_TEST BrbUaConvVariantValueToString_DateTime(void)
{
	memset(&variantIn0, 0, sizeof(variantIn0));
	variantIn0.VariantType = UAVariantType_DateTime;
	variantIn0.DateTime = BrbSetDt(2106, 02, 07, 06, 28, 15);
	dwordOut = BrbUaConvVariantValueToString(&variantIn0, stringIn0, sizeof(stringIn0));
	TEST_ASSERT_EQUAL_INT(0x00000000, dwordOut); // = Good
	BRB_ASSERT_EQUAL_DINT(UAVariantType_DateTime, (DINT)variantIn0.VariantType);
	TEST_ASSERT_EQUAL_STRING("2106-02-07 06:28:15", stringIn0);

	// Finished
	TEST_DONE;
}

_TEST BrbUaConvVariantValueToString_Guid(void)
{
	memset(&variantIn0, 0, sizeof(variantIn0));
	variantIn0.VariantType = UAVariantType_Guid;
	strcpy(variantIn0.String, "12345678-1234-5678-9ABC-123456789ABC");
	dwordOut = BrbUaConvVariantValueToString(&variantIn0, stringIn0, sizeof(stringIn0));
	TEST_ASSERT_EQUAL_INT(0x00000000, dwordOut); // = Good
	BRB_ASSERT_EQUAL_DINT(UAVariantType_Guid, (DINT)variantIn0.VariantType);
	TEST_ASSERT_EQUAL_STRING("12345678-1234-5678-9ABC-123456789ABC", stringIn0);

	// Finished
	TEST_DONE;
}

_TEST BrbUaConvVariantValueToString_ByteString(void)
{
	memset(&variantIn0, 0, sizeof(variantIn0));
	variantIn0.VariantType = UAVariantType_ByteString;
	dwordOut = BrbUaConvVariantValueToString(&variantIn0, stringIn0, sizeof(stringIn0));
	TEST_ASSERT_EQUAL_INT(0x803D0000, dwordOut); // = Bad_NotSupported
	BRB_ASSERT_EQUAL_DINT(UAVariantType_ByteString, (DINT)variantIn0.VariantType);

	// Finished
	TEST_DONE;
}

_TEST BrbUaConvVariantValueToString_XmlElement(void)
{
	memset(&variantIn0, 0, sizeof(variantIn0));
	variantIn0.VariantType = UAVariantType_XmlElement;
	dwordOut = BrbUaConvVariantValueToString(&variantIn0, stringIn0, sizeof(stringIn0));
	TEST_ASSERT_EQUAL_INT(0x803D0000, dwordOut); // = Bad_NotSupported
	BRB_ASSERT_EQUAL_DINT(UAVariantType_XmlElement, (DINT)variantIn0.VariantType);

	// Finished
	TEST_DONE;
}

_TEST BrbUaConvVariantValueToString_NodeId(void)
{
	memset(&variantIn0, 0, sizeof(variantIn0));
	variantIn0.VariantType = UAVariantType_NodeId;
	BrbUaSetNodeId(&variantIn0.NodeId, "VarX", 0);
	dwordOut = BrbUaConvVariantValueToString(&variantIn0, stringIn0, sizeof(stringIn0));
	TEST_ASSERT_EQUAL_INT(0x00000000, dwordOut); // = Good
	BRB_ASSERT_EQUAL_DINT(UAVariantType_NodeId, (DINT)variantIn0.VariantType);
	TEST_ASSERT_EQUAL_STRING("ns=0;s=VarX", stringIn0);

	memset(&variantIn0, 0, sizeof(variantIn0));
	variantIn0.VariantType = UAVariantType_NodeId;
	BrbUaSetNodeId(&variantIn0.NodeId, "1234", 1);
	dwordOut = BrbUaConvVariantValueToString(&variantIn0, stringIn0, sizeof(stringIn0));
	TEST_ASSERT_EQUAL_INT(0x00000000, dwordOut); // = Good
	BRB_ASSERT_EQUAL_DINT(UAVariantType_NodeId, (DINT)variantIn0.VariantType);
	TEST_ASSERT_EQUAL_STRING("ns=1;i=1234", stringIn0);

	memset(&variantIn0, 0, sizeof(variantIn0));
	variantIn0.VariantType = UAVariantType_NodeId;
	variantIn0.NodeId.IdentifierType = UAIdentifierType_GUID;
	strcpy(variantIn0.NodeId.Identifier, "12345678-1234-5678-9ABC-123456789ABC");
	variantIn0.NodeId.NamespaceIndex = 2;
	dwordOut = BrbUaConvVariantValueToString(&variantIn0, stringIn0, sizeof(stringIn0));
	TEST_ASSERT_EQUAL_INT(0x00000000, dwordOut); // = Good
	BRB_ASSERT_EQUAL_DINT(UAVariantType_NodeId, (DINT)variantIn0.VariantType);
	TEST_ASSERT_EQUAL_STRING("ns=2;g=12345678-1234-5678-9ABC-123456789ABC", stringIn0);

	memset(&variantIn0, 0, sizeof(variantIn0));
	variantIn0.VariantType = UAVariantType_NodeId;
	variantIn0.NodeId.IdentifierType = UAIdentifierType_Opaque;
	strcpy(variantIn0.NodeId.Identifier, "");
	variantIn0.NodeId.NamespaceIndex = 2;
	dwordOut = BrbUaConvVariantValueToString(&variantIn0, stringIn0, sizeof(stringIn0));
	TEST_ASSERT_EQUAL_INT(0x803D0000, dwordOut); // = Bad_NotSupported
	BRB_ASSERT_EQUAL_DINT(UAVariantType_NodeId, (DINT)variantIn0.VariantType);

	// Finished
	TEST_DONE;
}

_TEST BrbUaConvVariantValueToString_ExpandedNodeId(void)
{
	memset(&variantIn0, 0, sizeof(variantIn0));
	variantIn0.VariantType = UAVariantType_ExpandedNodeId;
	dwordOut = BrbUaConvVariantValueToString(&variantIn0, stringIn0, sizeof(stringIn0));
	TEST_ASSERT_EQUAL_INT(0x803D0000, dwordOut); // = Bad_NotSupported
	BRB_ASSERT_EQUAL_DINT(UAVariantType_ExpandedNodeId, (DINT)variantIn0.VariantType);

	// Finished
	TEST_DONE;
}

_TEST BrbUaConvVariantValueToString_StatusCode(void)
{
	memset(&variantIn0, 0, sizeof(variantIn0));
	variantIn0.VariantType = UAVariantType_StatusCode;
	variantIn0.UInt32 = 0x800D0000; // = Bad_ServerNotConnected
	dwordOut = BrbUaConvVariantValueToString(&variantIn0, stringIn0, sizeof(stringIn0));
	TEST_ASSERT_EQUAL_INT(0x00000000, dwordOut); // = Good
	BRB_ASSERT_EQUAL_DINT(UAVariantType_StatusCode, (DINT)variantIn0.VariantType);
	TEST_ASSERT_EQUAL_STRING("0x800D0000 = Bad_ServerNotConnected", stringIn0);

	// Finished
	TEST_DONE;
}

_TEST BrbUaConvVariantValueToString_QualifiedName(void)
{
	memset(&variantIn0, 0, sizeof(variantIn0));
	variantIn0.VariantType = UAVariantType_QualifiedName;
	BrbUaSetQualifedName(&variantIn0.QualifiedName, 1, "VarX");
	dwordOut = BrbUaConvVariantValueToString(&variantIn0, stringIn0, sizeof(stringIn0));
	TEST_ASSERT_EQUAL_INT(0x00000000, dwordOut); // = Good
	BRB_ASSERT_EQUAL_DINT(UAVariantType_QualifiedName, (DINT)variantIn0.VariantType);
	TEST_ASSERT_EQUAL_STRING("1:VarX", stringIn0);

	// Finished
	TEST_DONE;
}

_TEST BrbUaConvVariantValueToString_LocalizedText(void)
{
	memset(&variantIn0, 0, sizeof(variantIn0));
	variantIn0.VariantType = UAVariantType_LocalizedText;
	BrbUaSetLocalizedText(&variantIn0.LocalizedText, "", "VarX");
	dwordOut = BrbUaConvVariantValueToString(&variantIn0, stringIn0, sizeof(stringIn0));
	TEST_ASSERT_EQUAL_INT(0x00000000, dwordOut); // = Good
	BRB_ASSERT_EQUAL_DINT(UAVariantType_LocalizedText, (DINT)variantIn0.VariantType);
	TEST_ASSERT_EQUAL_STRING("VarX", stringIn0);

	memset(&variantIn0, 0, sizeof(variantIn0));
	variantIn0.VariantType = UAVariantType_LocalizedText;
	BrbUaSetLocalizedText(&variantIn0.LocalizedText, "de", "VarX");
	dwordOut = BrbUaConvVariantValueToString(&variantIn0, stringIn0, sizeof(stringIn0));
	TEST_ASSERT_EQUAL_INT(0x00000000, dwordOut); // = Good
	BRB_ASSERT_EQUAL_DINT(UAVariantType_LocalizedText, (DINT)variantIn0.VariantType);
	TEST_ASSERT_EQUAL_STRING("de:VarX", stringIn0);

	// Finished
	TEST_DONE;
}

// NOLINTEND(readability-*, bugprone-easily-swappable-parameters, bugprone-branch-clone, clang-diagnostic-invalid-utf8, clang-diagnostic-invalid-source-encoding, clang-diagnostic-pointer-arith, clang-diagnostic-strict-prototypes, clang-diagnostic-bad-function-cast, clang-analyzer-security.insecureAPI.*, hicpp-uppercase-literal-suffix, cppcoreguidelines-*, performance-*)

/*
B+R UnitTest: This is generated code.
Do not edit! Do not move!
Description: UnitTest Testprogramm infrastructure (TestSet).
LastUpdated: 2023-05-05 10:56:29Z
By B+R UnitTest Helper Version: 2.0.1.59
*/
UNITTEST_FIXTURES(fixtures)
{
	new_TestFixture("BrbUaConvVariantValueToString_NulPtr", BrbUaConvVariantValueToString_NulPtr),
	new_TestFixture("BrbUaConvVariantValueToString_Bool", BrbUaConvVariantValueToString_Bool),
	new_TestFixture("BrbUaConvVariantValueToString_SByte", BrbUaConvVariantValueToString_SByte),
	new_TestFixture("BrbUaConvVariantValueToString_Byte", BrbUaConvVariantValueToString_Byte),
	new_TestFixture("BrbUaConvVariantValueToString_Int16", BrbUaConvVariantValueToString_Int16),
	new_TestFixture("BrbUaConvVariantValueToString_UInt16", BrbUaConvVariantValueToString_UInt16),
	new_TestFixture("BrbUaConvVariantValueToString_Int32", BrbUaConvVariantValueToString_Int32),
	new_TestFixture("BrbUaConvVariantValueToString_UInt32", BrbUaConvVariantValueToString_UInt32),
	new_TestFixture("BrbUaConvVariantValueToString_Int64", BrbUaConvVariantValueToString_Int64),
	new_TestFixture("BrbUaConvVariantValueToString_UInt64", BrbUaConvVariantValueToString_UInt64),
	new_TestFixture("BrbUaConvVariantValueToString_Float", BrbUaConvVariantValueToString_Float),
	new_TestFixture("BrbUaConvVariantValueToString_Double", BrbUaConvVariantValueToString_Double),
	new_TestFixture("BrbUaConvVariantValueToString_String", BrbUaConvVariantValueToString_String),
	new_TestFixture("BrbUaConvVariantValueToString_DateTime", BrbUaConvVariantValueToString_DateTime),
	new_TestFixture("BrbUaConvVariantValueToString_Guid", BrbUaConvVariantValueToString_Guid),
	new_TestFixture("BrbUaConvVariantValueToString_ByteString", BrbUaConvVariantValueToString_ByteString),
	new_TestFixture("BrbUaConvVariantValueToString_XmlElement", BrbUaConvVariantValueToString_XmlElement),
	new_TestFixture("BrbUaConvVariantValueToString_NodeId", BrbUaConvVariantValueToString_NodeId),
	new_TestFixture("BrbUaConvVariantValueToString_ExpandedNodeId", BrbUaConvVariantValueToString_ExpandedNodeId),
	new_TestFixture("BrbUaConvVariantValueToString_StatusCode", BrbUaConvVariantValueToString_StatusCode),
	new_TestFixture("BrbUaConvVariantValueToString_QualifiedName", BrbUaConvVariantValueToString_QualifiedName),
	new_TestFixture("BrbUaConvVariantValueToString_LocalizedText", BrbUaConvVariantValueToString_LocalizedText),
};

UNITTEST_CALLER_COMPLETE_EXPLICIT(Set_BrbUaConvVariantValueToString, "Set_BrbUaConvVariantValueToString", 0, 0, fixtures, 0, 0, 0);
```

#### Set_BrbUaAddVariantValueSubName.c - Test set
```c
#include <bur/plctypes.h>

#ifdef _DEFAULT_INCLUDES
#include <AsDefault.h>
#endif

#include "UnitTest.h"
#include "BrbAsserts.h"
#include <string.h>

// NOLINTBEGIN(readability-*, bugprone-easily-swappable-parameters, bugprone-branch-clone, clang-diagnostic-invalid-utf8, clang-diagnostic-invalid-source-encoding, clang-diagnostic-pointer-arith, clang-diagnostic-strict-prototypes, clang-diagnostic-bad-function-cast, clang-analyzer-security.insecureAPI.*, hicpp-uppercase-literal-suffix, cppcoreguidelines-*, performance-*)

_TEST BrbUaAddVariantValueSubName_NulPtr(void)
{
	dwordOut = BrbUaAddVariantValueSubName(0, 0, sizeof(stringIn0));
	TEST_ASSERT_EQUAL_INT(0x80460000, dwordOut); // = Bad_StructureMissing

	// Finished
	TEST_DONE;
}

_TEST BrbUaAddVariantValueSubName_Add(void)
{
	strcpy(stringIn0, "Var");
	dwordOut = BrbUaAddVariantValueSubName(UAVariantType_Null, stringIn0, sizeof(stringIn0));
	TEST_ASSERT_EQUAL_INT(0x803D0000, dwordOut); // = Bad_NotSupported

	strcpy(stringIn0, "Var");
	dwordOut = BrbUaAddVariantValueSubName(UAVariantType_Boolean, stringIn0, sizeof(stringIn0));
	TEST_ASSERT_EQUAL_INT(0x00000000, dwordOut); // = Good
	TEST_ASSERT_EQUAL_STRING("Var.Boolean", stringIn0);

	strcpy(stringIn0, "Var");
	dwordOut = BrbUaAddVariantValueSubName(UAVariantType_SByte, stringIn0, sizeof(stringIn0));
	TEST_ASSERT_EQUAL_INT(0x00000000, dwordOut); // = Good
	TEST_ASSERT_EQUAL_STRING("Var.SByte", stringIn0);

	strcpy(stringIn0, "Var");
	dwordOut = BrbUaAddVariantValueSubName(UAVariantType_Byte, stringIn0, sizeof(stringIn0));
	TEST_ASSERT_EQUAL_INT(0x00000000, dwordOut); // = Good
	TEST_ASSERT_EQUAL_STRING("Var.Byte", stringIn0);

	strcpy(stringIn0, "Var");
	dwordOut = BrbUaAddVariantValueSubName(UAVariantType_Int16, stringIn0, sizeof(stringIn0));
	TEST_ASSERT_EQUAL_INT(0x00000000, dwordOut); // = Good
	TEST_ASSERT_EQUAL_STRING("Var.Int16", stringIn0);

	strcpy(stringIn0, "Var");
	dwordOut = BrbUaAddVariantValueSubName(UAVariantType_UInt16, stringIn0, sizeof(stringIn0));
	TEST_ASSERT_EQUAL_INT(0x00000000, dwordOut); // = Good
	TEST_ASSERT_EQUAL_STRING("Var.UInt16", stringIn0);

	strcpy(stringIn0, "Var");
	dwordOut = BrbUaAddVariantValueSubName(UAVariantType_Int32, stringIn0, sizeof(stringIn0));
	TEST_ASSERT_EQUAL_INT(0x00000000, dwordOut); // = Good
	TEST_ASSERT_EQUAL_STRING("Var.Int32", stringIn0);

	strcpy(stringIn0, "Var");
	dwordOut = BrbUaAddVariantValueSubName(UAVariantType_UInt32, stringIn0, sizeof(stringIn0));
	TEST_ASSERT_EQUAL_INT(0x00000000, dwordOut); // = Good
	TEST_ASSERT_EQUAL_STRING("Var.UInt32", stringIn0);

	strcpy(stringIn0, "Var");
	dwordOut = BrbUaAddVariantValueSubName(UAVariantType_Int64, stringIn0, sizeof(stringIn0));
	TEST_ASSERT_EQUAL_INT(0x00000000, dwordOut); // = Good
	TEST_ASSERT_EQUAL_STRING("Var.Int64", stringIn0);

	strcpy(stringIn0, "Var");
	dwordOut = BrbUaAddVariantValueSubName(UAVariantType_UInt64, stringIn0, sizeof(stringIn0));
	TEST_ASSERT_EQUAL_INT(0x00000000, dwordOut); // = Good
	TEST_ASSERT_EQUAL_STRING("Var.UInt64", stringIn0);

	strcpy(stringIn0, "Var");
	dwordOut = BrbUaAddVariantValueSubName(UAVariantType_Float, stringIn0, sizeof(stringIn0));
	TEST_ASSERT_EQUAL_INT(0x00000000, dwordOut); // = Good
	TEST_ASSERT_EQUAL_STRING("Var.Float", stringIn0);

	strcpy(stringIn0, "Var");
	dwordOut = BrbUaAddVariantValueSubName(UAVariantType_Double, stringIn0, sizeof(stringIn0));
	TEST_ASSERT_EQUAL_INT(0x00000000, dwordOut); // = Good
	TEST_ASSERT_EQUAL_STRING("Var.Double", stringIn0);

	strcpy(stringIn0, "Var");
	dwordOut = BrbUaAddVariantValueSubName(UAVariantType_String, stringIn0, sizeof(stringIn0));
	TEST_ASSERT_EQUAL_INT(0x00000000, dwordOut); // = Good
	TEST_ASSERT_EQUAL_STRING("Var.String", stringIn0);

	strcpy(stringIn0, "Var");
	dwordOut = BrbUaAddVariantValueSubName(UAVariantType_DateTime, stringIn0, sizeof(stringIn0));
	TEST_ASSERT_EQUAL_INT(0x00000000, dwordOut); // = Good
	TEST_ASSERT_EQUAL_STRING("Var.DateTime", stringIn0);

	strcpy(stringIn0, "Var");
	dwordOut = BrbUaAddVariantValueSubName(UAVariantType_Guid, stringIn0, sizeof(stringIn0));
	TEST_ASSERT_EQUAL_INT(0x00000000, dwordOut); // = Good
	TEST_ASSERT_EQUAL_STRING("Var.String", stringIn0);

	strcpy(stringIn0, "Var");
	dwordOut = BrbUaAddVariantValueSubName(UAVariantType_ByteString, stringIn0, sizeof(stringIn0));
	TEST_ASSERT_EQUAL_INT(0x00000000, dwordOut); // = Good
	TEST_ASSERT_EQUAL_STRING("Var.String", stringIn0);

	strcpy(stringIn0, "Var");
	dwordOut = BrbUaAddVariantValueSubName(UAVariantType_XmlElement, stringIn0, sizeof(stringIn0));
	TEST_ASSERT_EQUAL_INT(0x803D0000, dwordOut); // = Bad_NotSupported

	strcpy(stringIn0, "Var");
	dwordOut = BrbUaAddVariantValueSubName(UAVariantType_NodeId, stringIn0, sizeof(stringIn0));
	TEST_ASSERT_EQUAL_INT(0x00000000, dwordOut); // = Good
	TEST_ASSERT_EQUAL_STRING("Var.NodeId", stringIn0);

	strcpy(stringIn0, "Var");
	dwordOut = BrbUaAddVariantValueSubName(UAVariantType_ExpandedNodeId, stringIn0, sizeof(stringIn0));
	TEST_ASSERT_EQUAL_INT(0x00000000, dwordOut); // = Good
	TEST_ASSERT_EQUAL_STRING("Var.ExpandedNodeId", stringIn0);

	strcpy(stringIn0, "Var");
	dwordOut = BrbUaAddVariantValueSubName(UAVariantType_StatusCode, stringIn0, sizeof(stringIn0));
	TEST_ASSERT_EQUAL_INT(0x00000000, dwordOut); // = Good
	TEST_ASSERT_EQUAL_STRING("Var.StatusCode", stringIn0);

	strcpy(stringIn0, "Var");
	dwordOut = BrbUaAddVariantValueSubName(UAVariantType_QualifiedName, stringIn0, sizeof(stringIn0));
	TEST_ASSERT_EQUAL_INT(0x00000000, dwordOut); // = Good
	TEST_ASSERT_EQUAL_STRING("Var.QualifiedName", stringIn0);

	strcpy(stringIn0, "Var");
	dwordOut = BrbUaAddVariantValueSubName(UAVariantType_Boolean, stringIn0, sizeof(stringIn0));
	TEST_ASSERT_EQUAL_INT(0x00000000, dwordOut); // = Good
	TEST_ASSERT_EQUAL_STRING("Var.Boolean", stringIn0);

	strcpy(stringIn0, "Var");
	dwordOut = BrbUaAddVariantValueSubName(UAVariantType_LocalizedText, stringIn0, sizeof(stringIn0));
	TEST_ASSERT_EQUAL_INT(0x00000000, dwordOut); // = Good
	TEST_ASSERT_EQUAL_STRING("Var.LocalizedText", stringIn0);

	// Finished
	TEST_DONE;
}

// NOLINTEND(readability-*, bugprone-easily-swappable-parameters, bugprone-branch-clone, clang-diagnostic-invalid-utf8, clang-diagnostic-invalid-source-encoding, clang-diagnostic-pointer-arith, clang-diagnostic-strict-prototypes, clang-diagnostic-bad-function-cast, clang-analyzer-security.insecureAPI.*, hicpp-uppercase-literal-suffix, cppcoreguidelines-*, performance-*)

/*
B+R UnitTest: This is generated code.
Do not edit! Do not move!
Description: UnitTest Testprogramm infrastructure (TestSet).
LastUpdated: 2023-04-20 12:30:26Z
By B+R UnitTest Helper Version: 2.0.1.59
*/
UNITTEST_FIXTURES(fixtures)
{
	new_TestFixture("BrbUaAddVariantValueSubName_NulPtr", BrbUaAddVariantValueSubName_NulPtr),
	new_TestFixture("BrbUaAddVariantValueSubName_Add", BrbUaAddVariantValueSubName_Add),
};

UNITTEST_CALLER_COMPLETE_EXPLICIT(Set_BrbUaAddVariantValueSubName, "Set_BrbUaAddVariantValueSubName", 0, 0, fixtures, 0, 0, 0);
```

### Program Logical/UnitTests/UtBrbLibUa/UtBrbUaByteStrings (ANSIC) - UnitTests

#### variables.var - Name the suite and add PVs for the program
```iecst
(********************************************************************
 * COPYRIGHT --
 ********************************************************************
 * Program: utTemplate_automated
 * File: variables.var
 * Author: -
 * Created: -
 ********************************************************************
 * Local variables of program utTemplate_automated
 ********************************************************************)
(*Describe the test*)
VAR
	Testsuite : UtMgrTestSuite := (Name:='BrbUaByteStrings',Description:='(Optional field)Template for use with helper tool. Reference or add this program in the package "TS_UnitTest_UpdateTestPrograms"',Type:=utMgrTEST_TYPE_C,MetaInformation:='(Optional field):To be filled');
END_VAR
(*Input variables for testing*)
(*Constants*)
VAR CONSTANT
	nBYTE_STRING_INDEX_MAX : UINT := 4;
END_VAR
VAR
	byteStringIn : ARRAY[0..nBYTE_STRING_INDEX_MAX] OF USINT;
END_VAR
(*Functionblock instances for testing*)
(*Output variables for testing*)
VAR
	dwordOut : DWORD;
END_VAR
```

#### autoGeneratedFile.c - Auto generated code - list of all test sets in the program
```c
/*
B+R UnitTest: This is generated code.
Do not edit! Do not move!
Description: UnitTest Testprogramm infrastructure (List of TestSets).
LastUpdated: 2023-04-25 07:04:32Z
By B+R UnitTest Helper Version: 2.0.1.59
*/
#include "UnitTest.h"

UNITTEST_TESTSET_DECLARATION  Set_BrbUaIncByteString;
UNITTEST_TESTSET_DECLARATION  Set_BrbUaGetRandomByteString;

UNITTEST_TESTSET_FIXTURES(utTestSets)
{
	new_TestSet(Set_BrbUaIncByteString),
	new_TestSet(Set_BrbUaGetRandomByteString),
};
UNTITTEST_TESTSET_HANDLER();
```

#### Set_BrbUaIncByteString.c - Test set
```c
#include <bur/plctypes.h>

#ifdef _DEFAULT_INCLUDES
#include <AsDefault.h>
#endif

#include "UnitTest.h"
#include "BrbAsserts.h"
#include <string.h>

// NOLINTBEGIN(readability-*, bugprone-easily-swappable-parameters, bugprone-branch-clone, clang-diagnostic-invalid-utf8, clang-diagnostic-invalid-source-encoding, clang-diagnostic-pointer-arith, clang-diagnostic-strict-prototypes, clang-diagnostic-bad-function-cast, clang-analyzer-security.insecureAPI.*, hicpp-uppercase-literal-suffix, cppcoreguidelines-*, performance-*)
_TEST BrbUaIncByteString_NulPtr(void)
{
	dwordOut = BrbUaIncByteString(0, 0);
	TEST_ASSERT_EQUAL_INT(0x80460000, dwordOut); // = Bad_StructureMissing

	// Finished
	TEST_DONE;
}

_TEST BrbUaIncByteString_Inc(void)
{
	memset(&byteStringIn, 1, sizeof(byteStringIn));
	dwordOut = BrbUaIncByteString((USINT*)&byteStringIn, 0);
	TEST_ASSERT_EQUAL_INT(0x803C0000, dwordOut); // = Bad_OutOfRange

	memset(&byteStringIn, 0, sizeof(byteStringIn));
	dwordOut = BrbUaIncByteString((USINT*)&byteStringIn, nBYTE_STRING_INDEX_MAX+1);
	TEST_ASSERT_EQUAL_INT(0x00000000, dwordOut); // = Good
	BRB_ASSERT_EQUAL_UDINT(0, (UDINT)byteStringIn[0]);
	BRB_ASSERT_EQUAL_UDINT(0, (UDINT)byteStringIn[1]);
	BRB_ASSERT_EQUAL_UDINT(0, (UDINT)byteStringIn[2]);
	BRB_ASSERT_EQUAL_UDINT(0, (UDINT)byteStringIn[3]);
	BRB_ASSERT_EQUAL_UDINT(1, (UDINT)byteStringIn[4]);

	dwordOut = BrbUaIncByteString((USINT*)&byteStringIn, nBYTE_STRING_INDEX_MAX+1);
	TEST_ASSERT_EQUAL_INT(0x00000000, dwordOut); // = Good
	BRB_ASSERT_EQUAL_UDINT(0, (UDINT)byteStringIn[0]);
	BRB_ASSERT_EQUAL_UDINT(0, (UDINT)byteStringIn[1]);
	BRB_ASSERT_EQUAL_UDINT(0, (UDINT)byteStringIn[2]);
	BRB_ASSERT_EQUAL_UDINT(0, (UDINT)byteStringIn[3]);
	BRB_ASSERT_EQUAL_UDINT(2, (UDINT)byteStringIn[4]);

	byteStringIn[0] = 0;
	byteStringIn[1] = 0;
	byteStringIn[2] = 0;
	byteStringIn[3] = 0;
	byteStringIn[4] = 255;
	dwordOut = BrbUaIncByteString((USINT*)&byteStringIn, nBYTE_STRING_INDEX_MAX+1);
	TEST_ASSERT_EQUAL_INT(0x00000000, dwordOut); // = Good
	BRB_ASSERT_EQUAL_UDINT(0, (UDINT)byteStringIn[0]);
	BRB_ASSERT_EQUAL_UDINT(0, (UDINT)byteStringIn[1]);
	BRB_ASSERT_EQUAL_UDINT(0, (UDINT)byteStringIn[2]);
	BRB_ASSERT_EQUAL_UDINT(1, (UDINT)byteStringIn[3]);
	BRB_ASSERT_EQUAL_UDINT(0, (UDINT)byteStringIn[4]);

	byteStringIn[0] = 0;
	byteStringIn[1] = 0;
	byteStringIn[2] = 0;
	byteStringIn[3] = 255;
	byteStringIn[4] = 255;
	dwordOut = BrbUaIncByteString((USINT*)&byteStringIn, nBYTE_STRING_INDEX_MAX+1);
	TEST_ASSERT_EQUAL_INT(0x00000000, dwordOut); // = Good
	BRB_ASSERT_EQUAL_UDINT(0, (UDINT)byteStringIn[0]);
	BRB_ASSERT_EQUAL_UDINT(0, (UDINT)byteStringIn[1]);
	BRB_ASSERT_EQUAL_UDINT(1, (UDINT)byteStringIn[2]);
	BRB_ASSERT_EQUAL_UDINT(0, (UDINT)byteStringIn[3]);
	BRB_ASSERT_EQUAL_UDINT(0, (UDINT)byteStringIn[4]);

	byteStringIn[0] = 0;
	byteStringIn[1] = 0;
	byteStringIn[2] = 255;
	byteStringIn[3] = 255;
	byteStringIn[4] = 255;
	dwordOut = BrbUaIncByteString((USINT*)&byteStringIn, nBYTE_STRING_INDEX_MAX+1);
	TEST_ASSERT_EQUAL_INT(0x00000000, dwordOut); // = Good
	BRB_ASSERT_EQUAL_UDINT(0, (UDINT)byteStringIn[0]);
	BRB_ASSERT_EQUAL_UDINT(1, (UDINT)byteStringIn[1]);
	BRB_ASSERT_EQUAL_UDINT(0, (UDINT)byteStringIn[2]);
	BRB_ASSERT_EQUAL_UDINT(0, (UDINT)byteStringIn[3]);
	BRB_ASSERT_EQUAL_UDINT(0, (UDINT)byteStringIn[4]);

	byteStringIn[0] = 0;
	byteStringIn[1] = 255;
	byteStringIn[2] = 255;
	byteStringIn[3] = 255;
	byteStringIn[4] = 255;
	dwordOut = BrbUaIncByteString((USINT*)&byteStringIn, nBYTE_STRING_INDEX_MAX+1);
	TEST_ASSERT_EQUAL_INT(0x00000000, dwordOut); // = Good
	BRB_ASSERT_EQUAL_UDINT(1, (UDINT)byteStringIn[0]);
	BRB_ASSERT_EQUAL_UDINT(0, (UDINT)byteStringIn[1]);
	BRB_ASSERT_EQUAL_UDINT(0, (UDINT)byteStringIn[2]);
	BRB_ASSERT_EQUAL_UDINT(0, (UDINT)byteStringIn[3]);
	BRB_ASSERT_EQUAL_UDINT(0, (UDINT)byteStringIn[4]);

	byteStringIn[0] = 255;
	byteStringIn[1] = 255;
	byteStringIn[2] = 255;
	byteStringIn[3] = 255;
	byteStringIn[4] = 255;
	dwordOut = BrbUaIncByteString((USINT*)&byteStringIn, nBYTE_STRING_INDEX_MAX+1);
	TEST_ASSERT_EQUAL_INT(0xB00C0000, dwordOut); // = PlcOpen_BadElementCount
	BRB_ASSERT_EQUAL_UDINT(0, (UDINT)byteStringIn[0]);
	BRB_ASSERT_EQUAL_UDINT(0, (UDINT)byteStringIn[1]);
	BRB_ASSERT_EQUAL_UDINT(0, (UDINT)byteStringIn[2]);
	BRB_ASSERT_EQUAL_UDINT(0, (UDINT)byteStringIn[3]);
	BRB_ASSERT_EQUAL_UDINT(0, (UDINT)byteStringIn[4]);

	// Finished
	TEST_DONE;
}

// NOLINTEND(readability-*, bugprone-easily-swappable-parameters, bugprone-branch-clone, clang-diagnostic-invalid-utf8, clang-diagnostic-invalid-source-encoding, clang-diagnostic-pointer-arith, clang-diagnostic-strict-prototypes, clang-diagnostic-bad-function-cast, clang-analyzer-security.insecureAPI.*, hicpp-uppercase-literal-suffix, cppcoreguidelines-*, performance-*)

/*
B+R UnitTest: This is generated code.
Do not edit! Do not move!
Description: UnitTest Testprogramm infrastructure (TestSet).
LastUpdated: 2023-04-20 12:39:56Z
By B+R UnitTest Helper Version: 2.0.1.59
*/
UNITTEST_FIXTURES(fixtures)
{
	new_TestFixture("BrbUaIncByteString_NulPtr", BrbUaIncByteString_NulPtr),
	new_TestFixture("BrbUaIncByteString_Inc", BrbUaIncByteString_Inc),
};

UNITTEST_CALLER_COMPLETE_EXPLICIT(Set_BrbUaIncByteString, "Set_BrbUaIncByteString", 0, 0, fixtures, 0, 0, 0);
```

#### Set_BrbUaGetRandomByteString.c - Test set
```c
#include <bur/plctypes.h>

#ifdef _DEFAULT_INCLUDES
#include <AsDefault.h>
#endif

#include "UnitTest.h"
#include "BrbAsserts.h"
#include <string.h>

// NOLINTBEGIN(readability-*, bugprone-easily-swappable-parameters, bugprone-branch-clone, clang-diagnostic-invalid-utf8, clang-diagnostic-invalid-source-encoding, clang-diagnostic-pointer-arith, clang-diagnostic-strict-prototypes, clang-diagnostic-bad-function-cast, clang-analyzer-security.insecureAPI.*, hicpp-uppercase-literal-suffix, cppcoreguidelines-*, performance-*)
_TEST BrbUaGetRandomByteString_NulPtr(void)
{
	dwordOut = BrbUaGetRandomByteString(0, 0);
	TEST_ASSERT_EQUAL_INT(0x80460000, dwordOut); // = Bad_StructureMissing

	// Finished
	TEST_DONE;
}

_TEST BrbUaGetRandomByteString_Random(void)
{
	dwordOut = BrbUaGetRandomByteString((USINT*)&byteStringIn, 0);
	TEST_ASSERT_EQUAL_INT(0x803C0000, dwordOut); // = Bad_OutOfRange

	dwordOut = BrbUaGetRandomByteString((USINT*)&byteStringIn, nBYTE_STRING_INDEX_MAX+1);
	TEST_ASSERT_EQUAL_INT(0x00000000, dwordOut); // = Good

	// Finished
	TEST_DONE;
}

// NOLINTEND(readability-*, bugprone-easily-swappable-parameters, bugprone-branch-clone, clang-diagnostic-invalid-utf8, clang-diagnostic-invalid-source-encoding, clang-diagnostic-pointer-arith, clang-diagnostic-strict-prototypes, clang-diagnostic-bad-function-cast, clang-analyzer-security.insecureAPI.*, hicpp-uppercase-literal-suffix, cppcoreguidelines-*, performance-*)

/*
B+R UnitTest: This is generated code.
Do not edit! Do not move!
Description: UnitTest Testprogramm infrastructure (TestSet).
LastUpdated: 2023-04-25 07:04:32Z
By B+R UnitTest Helper Version: 2.0.1.59
*/
UNITTEST_FIXTURES(fixtures)
{
	new_TestFixture("BrbUaGetRandomByteString_NulPtr", BrbUaGetRandomByteString_NulPtr),
	new_TestFixture("BrbUaGetRandomByteString_Random", BrbUaGetRandomByteString_Random),
};

UNITTEST_CALLER_COMPLETE_EXPLICIT(Set_BrbUaGetRandomByteString, "Set_BrbUaGetRandomByteString", 0, 0, fixtures, 0, 0, 0);
```

### Program Logical/UnitTests/UtBrbLibUa/UtBrbUaLocalizedTexts (ANSIC) - UnitTests

#### variables.var - Name the suite and add PVs for the program
```iecst
(********************************************************************
 * COPYRIGHT --
 ********************************************************************
 * Program: utTemplate_automated
 * File: variables.var
 * Author: -
 * Created: -
 ********************************************************************
 * Local variables of program utTemplate_automated
 ********************************************************************)
(*Describe the test*)
VAR
	Testsuite : UtMgrTestSuite := (Name:='BrbUaLocalizedTexts',Description:='(Optional field)Template for use with helper tool. Reference or add this program in the package "TS_UnitTest_UpdateTestPrograms"',Type:=utMgrTEST_TYPE_C,MetaInformation:='(Optional field):To be filled');
END_VAR
(*Input variables for testing*)
(*Constants*)
VAR
	localizedTextIn : BrUaLocalizedText;
	stringIn : STRING[32];
END_VAR
(*Functionblock instances for testing*)
(*Output variables for testing*)
VAR
	dwordOut : DWORD;
END_VAR
```

#### autoGeneratedFile.c - Auto generated code - list of all test sets in the program
```c
/*
B+R UnitTest: This is generated code.
Do not edit! Do not move!
Description: UnitTest Testprogramm infrastructure (List of TestSets).
LastUpdated: 2023-04-25 07:20:13Z
By B+R UnitTest Helper Version: 2.0.1.59
*/
#include "UnitTest.h"

UNITTEST_TESTSET_DECLARATION  Set_BrbUaSetLocalizedText;
UNITTEST_TESTSET_DECLARATION  Set_BrbUaGetRandomLocalizedText;
UNITTEST_TESTSET_DECLARATION  Set_BrbUaAddLocalizedTextText;

UNITTEST_TESTSET_FIXTURES(utTestSets)
{
	new_TestSet(Set_BrbUaSetLocalizedText),
	new_TestSet(Set_BrbUaGetRandomLocalizedText),
	new_TestSet(Set_BrbUaAddLocalizedTextText),
};
UNTITTEST_TESTSET_HANDLER();
```

#### Set_BrbUaSetLocalizedText.c - Test set
```c
#include <bur/plctypes.h>

#ifdef _DEFAULT_INCLUDES
#include <AsDefault.h>
#endif

#include "UnitTest.h"
#include "BrbAsserts.h"
#include <string.h>

// NOLINTBEGIN(readability-*, bugprone-easily-swappable-parameters, bugprone-branch-clone, clang-diagnostic-invalid-utf8, clang-diagnostic-invalid-source-encoding, clang-diagnostic-pointer-arith, clang-diagnostic-strict-prototypes, clang-diagnostic-bad-function-cast, clang-analyzer-security.insecureAPI.*, hicpp-uppercase-literal-suffix, cppcoreguidelines-*, performance-*)
_TEST BrbUaSetLocalizedText_NulPtr(void)
{
	dwordOut = BrbUaSetLocalizedText(0, "de", "Hello");
	TEST_ASSERT_EQUAL_INT(0x80460000, dwordOut); // = Bad_StructureMissing

	dwordOut = BrbUaSetLocalizedText(&localizedTextIn, 0, "Hello");
	TEST_ASSERT_EQUAL_INT(0x80460000, dwordOut); // = Bad_StructureMissing

	dwordOut = BrbUaSetLocalizedText(&localizedTextIn, "de", 0);
	TEST_ASSERT_EQUAL_INT(0x80460000, dwordOut); // = Bad_StructureMissing

	// Finished
	TEST_DONE;
}

_TEST BrbUaSetLocalizedText_Set(void)
{
	dwordOut = BrbUaSetLocalizedText(&localizedTextIn, "de", "Hello");
	TEST_ASSERT_EQUAL_INT(0x00000000, dwordOut); // = Good
	TEST_ASSERT_EQUAL_STRING("de", localizedTextIn.Locale);
	TEST_ASSERT_EQUAL_STRING("Hello", localizedTextIn.Text);

	// Finished
	TEST_DONE;
}

// NOLINTEND(readability-*, bugprone-easily-swappable-parameters, bugprone-branch-clone, clang-diagnostic-invalid-utf8, clang-diagnostic-invalid-source-encoding, clang-diagnostic-pointer-arith, clang-diagnostic-strict-prototypes, clang-diagnostic-bad-function-cast, clang-analyzer-security.insecureAPI.*, hicpp-uppercase-literal-suffix, cppcoreguidelines-*, performance-*)

/*
B+R UnitTest: This is generated code.
Do not edit! Do not move!
Description: UnitTest Testprogramm infrastructure (TestSet).
LastUpdated: 2023-04-25 07:11:16Z
By B+R UnitTest Helper Version: 2.0.1.59
*/
UNITTEST_FIXTURES(fixtures)
{
	new_TestFixture("BrbUaSetLocalizedText_NulPtr", BrbUaSetLocalizedText_NulPtr),
	new_TestFixture("BrbUaSetLocalizedText_Set", BrbUaSetLocalizedText_Set),
};

UNITTEST_CALLER_COMPLETE_EXPLICIT(Set_BrbUaSetLocalizedText, "Set_BrbUaSetLocalizedText", 0, 0, fixtures, 0, 0, 0);
```

#### Set_BrbUaGetRandomLocalizedText.c - Test set
```c
#include <bur/plctypes.h>

#ifdef _DEFAULT_INCLUDES
#include <AsDefault.h>
#endif

#include "UnitTest.h"
#include "BrbAsserts.h"
#include <string.h>

// NOLINTBEGIN(readability-*, bugprone-easily-swappable-parameters, bugprone-branch-clone, clang-diagnostic-invalid-utf8, clang-diagnostic-invalid-source-encoding, clang-diagnostic-pointer-arith, clang-diagnostic-strict-prototypes, clang-diagnostic-bad-function-cast, clang-analyzer-security.insecureAPI.*, hicpp-uppercase-literal-suffix, cppcoreguidelines-*, performance-*)
_TEST BrbUaGetRandomLocalizedText_NulPtr(void)
{
	dwordOut = BrbUaGetRandomLocalizedText(0, 0);
	TEST_ASSERT_EQUAL_INT(0x80460000, dwordOut); // = Bad_StructureMissing

	// Finished
	TEST_DONE;
}

_TEST BrbUaGetRandomLocalizedText_Get(void)
{
	dwordOut = BrbUaGetRandomLocalizedText(&localizedTextIn, 10);
	TEST_ASSERT_EQUAL_INT(0x00000000, dwordOut); // = Good

	// Finished
	TEST_DONE;
}

// NOLINTEND(readability-*, bugprone-easily-swappable-parameters, bugprone-branch-clone, clang-diagnostic-invalid-utf8, clang-diagnostic-invalid-source-encoding, clang-diagnostic-pointer-arith, clang-diagnostic-strict-prototypes, clang-diagnostic-bad-function-cast, clang-analyzer-security.insecureAPI.*, hicpp-uppercase-literal-suffix, cppcoreguidelines-*, performance-*)

/*
B+R UnitTest: This is generated code.
Do not edit! Do not move!
Description: UnitTest Testprogramm infrastructure (TestSet).
LastUpdated: 2023-04-25 07:15:27Z
By B+R UnitTest Helper Version: 2.0.1.59
*/
UNITTEST_FIXTURES(fixtures)
{
	new_TestFixture("BrbUaGetRandomLocalizedText_NulPtr", BrbUaGetRandomLocalizedText_NulPtr),
	new_TestFixture("BrbUaGetRandomLocalizedText_Get", BrbUaGetRandomLocalizedText_Get),
};

UNITTEST_CALLER_COMPLETE_EXPLICIT(Set_BrbUaGetRandomLocalizedText, "Set_BrbUaGetRandomLocalizedText", 0, 0, fixtures, 0, 0, 0);
```

#### Set_BrbUaAddLocalizedTextText.c - Test set
```c
#include <bur/plctypes.h>

#ifdef _DEFAULT_INCLUDES
#include <AsDefault.h>
#endif

#include "UnitTest.h"
#include "BrbAsserts.h"
#include <string.h>

// NOLINTBEGIN(readability-*, bugprone-easily-swappable-parameters, bugprone-branch-clone, clang-diagnostic-invalid-utf8, clang-diagnostic-invalid-source-encoding, clang-diagnostic-pointer-arith, clang-diagnostic-strict-prototypes, clang-diagnostic-bad-function-cast, clang-analyzer-security.insecureAPI.*, hicpp-uppercase-literal-suffix, cppcoreguidelines-*, performance-*)
_TEST BrbUaAddLocalizedTextText_NulPtr(void)
{
	dwordOut = BrbUaAddLocalizedTextText(0, stringIn, sizeof(stringIn));
	TEST_ASSERT_EQUAL_INT(0x80460000, dwordOut); // = Bad_StructureMissing

	dwordOut = BrbUaAddLocalizedTextText(&localizedTextIn, 0, sizeof(stringIn));
	TEST_ASSERT_EQUAL_INT(0x80460000, dwordOut); // = Bad_StructureMissing

	// Finished
	TEST_DONE;
}

_TEST BrbUaAddLocalizedTextText_Add(void)
{
	strcpy(stringIn, "Test ");
	BrbUaSetLocalizedText(&localizedTextIn, "de", "Hello");
	dwordOut = BrbUaAddLocalizedTextText(&localizedTextIn, stringIn, sizeof(stringIn));
	TEST_ASSERT_EQUAL_INT(0x00000000, dwordOut); // = Good
	TEST_ASSERT_EQUAL_STRING("Test de:Hello", stringIn);

	strcpy(stringIn, "Test ");
	BrbUaSetLocalizedText(&localizedTextIn, "", "Hello");
	dwordOut = BrbUaAddLocalizedTextText(&localizedTextIn, stringIn, sizeof(stringIn));
	TEST_ASSERT_EQUAL_INT(0x00000000, dwordOut); // = Good
	TEST_ASSERT_EQUAL_STRING("Test Hello", stringIn);

	strcpy(stringIn, "Test ");
	BrbUaSetLocalizedText(&localizedTextIn, "en", "");
	dwordOut = BrbUaAddLocalizedTextText(&localizedTextIn, stringIn, sizeof(stringIn));
	TEST_ASSERT_EQUAL_INT(0x00000000, dwordOut); // = Good
	TEST_ASSERT_EQUAL_STRING("Test en:", stringIn);

	// Finished
	TEST_DONE;
}

// NOLINTEND(readability-*, bugprone-easily-swappable-parameters, bugprone-branch-clone, clang-diagnostic-invalid-utf8, clang-diagnostic-invalid-source-encoding, clang-diagnostic-pointer-arith, clang-diagnostic-strict-prototypes, clang-diagnostic-bad-function-cast, clang-analyzer-security.insecureAPI.*, hicpp-uppercase-literal-suffix, cppcoreguidelines-*, performance-*)

/*
B+R UnitTest: This is generated code.
Do not edit! Do not move!
Description: UnitTest Testprogramm infrastructure (TestSet).
LastUpdated: 2023-04-25 07:20:13Z
By B+R UnitTest Helper Version: 2.0.1.59
*/
UNITTEST_FIXTURES(fixtures)
{
	new_TestFixture("BrbUaAddLocalizedTextText_NulPtr", BrbUaAddLocalizedTextText_NulPtr),
	new_TestFixture("BrbUaAddLocalizedTextText_Add", BrbUaAddLocalizedTextText_Add),
};

UNITTEST_CALLER_COMPLETE_EXPLICIT(Set_BrbUaAddLocalizedTextText, "Set_BrbUaAddLocalizedTextText", 0, 0, fixtures, 0, 0, 0);
```

### Program Logical/UnitTests/UtBrbLibUa/UtBrbUaQualifiedNames (ANSIC) - UnitTests

#### variables.var - Name the suite and add PVs for the program
```iecst
(********************************************************************
 * COPYRIGHT --
 ********************************************************************
 * Program: utTemplate_automated
 * File: variables.var
 * Author: -
 * Created: -
 ********************************************************************
 * Local variables of program utTemplate_automated
 ********************************************************************)
(*Describe the test*)
VAR
	Testsuite : UtMgrTestSuite := (Name:='BrbUaQualifiedNames',Description:='(Optional field)Template for use with helper tool. Reference or add this program in the package "TS_UnitTest_UpdateTestPrograms"',Type:=utMgrTEST_TYPE_C,MetaInformation:='(Optional field):To be filled');
END_VAR
(*Input variables for testing*)
(*Constants*)
VAR
	qualifiedNameIn : BrUaQualifiedName;
END_VAR
(*Functionblock instances for testing*)
(*Output variables for testing*)
VAR
	dwordOut : DWORD;
END_VAR
```

#### autoGeneratedFile.c - Auto generated code - list of all test sets in the program
```c
/*
B+R UnitTest: This is generated code.
Do not edit! Do not move!
Description: UnitTest Testprogramm infrastructure (List of TestSets).
LastUpdated: 2023-04-25 07:27:30Z
By B+R UnitTest Helper Version: 2.0.1.59
*/
#include "UnitTest.h"

UNITTEST_TESTSET_DECLARATION  Set_BrbUaSetQualifiedName;
UNITTEST_TESTSET_DECLARATION  Set_BrbUaGetRandomQualifiedName;

UNITTEST_TESTSET_FIXTURES(utTestSets)
{
	new_TestSet(Set_BrbUaSetQualifiedName),
	new_TestSet(Set_BrbUaGetRandomQualifiedName),
};
UNTITTEST_TESTSET_HANDLER();
```

#### Set_BrbUaSetQualifiedName.c - Test set
```c
#include <bur/plctypes.h>

#ifdef _DEFAULT_INCLUDES
#include <AsDefault.h>
#endif

#include "UnitTest.h"
#include "BrbAsserts.h"
#include <string.h>

// NOLINTBEGIN(readability-*, bugprone-easily-swappable-parameters, bugprone-branch-clone, clang-diagnostic-invalid-utf8, clang-diagnostic-invalid-source-encoding, clang-diagnostic-pointer-arith, clang-diagnostic-strict-prototypes, clang-diagnostic-bad-function-cast, clang-analyzer-security.insecureAPI.*, hicpp-uppercase-literal-suffix, cppcoreguidelines-*, performance-*)
_TEST BrbUaSetQualifedName_NulPtr(void)
{
	dwordOut = BrbUaSetQualifedName(0, 1, "Hello");
	TEST_ASSERT_EQUAL_INT(0x80460000, dwordOut); // = Bad_StructureMissing

	dwordOut = BrbUaSetQualifedName(&qualifiedNameIn, 1, 0);
	TEST_ASSERT_EQUAL_INT(0x80460000, dwordOut); // = Bad_StructureMissing

	// Finished
	TEST_DONE;
}

_TEST BrbUaSetQualifedName_Set(void)
{
	dwordOut = BrbUaSetQualifedName(&qualifiedNameIn, 2, "Hello");
	TEST_ASSERT_EQUAL_INT(0x00000000, dwordOut); // = Good
	TEST_ASSERT_EQUAL_INT(2, qualifiedNameIn.NamespaceIndex);
	TEST_ASSERT_EQUAL_STRING("Hello", qualifiedNameIn.Name);

	// Finished
	TEST_DONE;
}

// NOLINTEND(readability-*, bugprone-easily-swappable-parameters, bugprone-branch-clone, clang-diagnostic-invalid-utf8, clang-diagnostic-invalid-source-encoding, clang-diagnostic-pointer-arith, clang-diagnostic-strict-prototypes, clang-diagnostic-bad-function-cast, clang-analyzer-security.insecureAPI.*, hicpp-uppercase-literal-suffix, cppcoreguidelines-*, performance-*)

/*
B+R UnitTest: This is generated code.
Do not edit! Do not move!
Description: UnitTest Testprogramm infrastructure (TestSet).
LastUpdated: 2023-04-25 07:25:45Z
By B+R UnitTest Helper Version: 2.0.1.59
*/
UNITTEST_FIXTURES(fixtures)
{
	new_TestFixture("BrbUaSetQualifedName_NulPtr", BrbUaSetQualifedName_NulPtr),
	new_TestFixture("BrbUaSetQualifedName_Set", BrbUaSetQualifedName_Set),
};

UNITTEST_CALLER_COMPLETE_EXPLICIT(Set_BrbUaSetQualifiedName, "Set_BrbUaSetQualifiedName", 0, 0, fixtures, 0, 0, 0);
```

#### Set_BrbUaGetRandomQualifiedName.c - Test set
```c
#include <bur/plctypes.h>

#ifdef _DEFAULT_INCLUDES
#include <AsDefault.h>
#endif

#include "UnitTest.h"
#include "BrbAsserts.h"
#include <string.h>

// NOLINTBEGIN(readability-*, bugprone-easily-swappable-parameters, bugprone-branch-clone, clang-diagnostic-invalid-utf8, clang-diagnostic-invalid-source-encoding, clang-diagnostic-pointer-arith, clang-diagnostic-strict-prototypes, clang-diagnostic-bad-function-cast, clang-analyzer-security.insecureAPI.*, hicpp-uppercase-literal-suffix, cppcoreguidelines-*, performance-*)
_TEST BrbUaGetRandomQualifiedName_NulPtr(void)
{
	dwordOut = BrbUaGetRandomQualifiedName(0, 0);
	TEST_ASSERT_EQUAL_INT(0x80460000, dwordOut); // = Bad_StructureMissing

	// Finished
	TEST_DONE;
}

_TEST BrbUaGetRandomQualifiedName_Get(void)
{
	dwordOut = BrbUaGetRandomQualifiedName(&qualifiedNameIn, 10);
	TEST_ASSERT_EQUAL_INT(0x00000000, dwordOut); // = Good

	// Finished
	TEST_DONE;
}

// NOLINTEND(readability-*, bugprone-easily-swappable-parameters, bugprone-branch-clone, clang-diagnostic-invalid-utf8, clang-diagnostic-invalid-source-encoding, clang-diagnostic-pointer-arith, clang-diagnostic-strict-prototypes, clang-diagnostic-bad-function-cast, clang-analyzer-security.insecureAPI.*, hicpp-uppercase-literal-suffix, cppcoreguidelines-*, performance-*)

/*
B+R UnitTest: This is generated code.
Do not edit! Do not move!
Description: UnitTest Testprogramm infrastructure (TestSet).
LastUpdated: 2023-04-25 07:27:30Z
By B+R UnitTest Helper Version: 2.0.1.59
*/
UNITTEST_FIXTURES(fixtures)
{
	new_TestFixture("BrbUaGetRandomQualifiedName_NulPtr", BrbUaGetRandomQualifiedName_NulPtr),
	new_TestFixture("BrbUaGetRandomQualifiedName_Get", BrbUaGetRandomQualifiedName_Get),
};

UNITTEST_CALLER_COMPLETE_EXPLICIT(Set_BrbUaGetRandomQualifiedName, "Set_BrbUaGetRandomQualifiedName", 0, 0, fixtures, 0, 0, 0);
```

### Program Logical/UnitTests/UtBrbLibUa/UtBrbUaTimeAndDate (ANSIC) - UnitTests

#### variables.var - Name the suite and add PVs for the program
```iecst
(********************************************************************
 * COPYRIGHT --
 ********************************************************************
 * Program: utTemplate_automated
 * File: variables.var
 * Author: -
 * Created: -
 ********************************************************************
 * Local variables of program utTemplate_automated
 ********************************************************************)
(*Describe the test*)
VAR
	Testsuite : UtMgrTestSuite := (Name:='BrbUaTimeAndDate',Description:='(Optional field)Template for use with helper tool. Reference or add this program in the package "TS_UnitTest_UpdateTestPrograms"',Type:=utMgrTEST_TYPE_C,MetaInformation:='(Optional field):To be filled');
END_VAR
(*Input variables for testing*)
(*Constants*)
VAR
	srvDateTimeIn : UaSrv_DateTimeType;
	dtStructIn : DTStructure;
	stringIn0 : STRING[64];
	stringIn1 : STRING[64];
	timeZoneDataIn : BrUaTimeZoneDataType;
END_VAR
(*Functionblock instances for testing*)
(*Output variables for testing*)
VAR
	uintOut : UINT;
	dwordOut : DWORD;
END_VAR
```

#### autoGeneratedFile.c - Auto generated code - list of all test sets in the program
```c
/*
B+R UnitTest: This is generated code.
Do not edit! Do not move!
Description: UnitTest Testprogramm infrastructure (List of TestSets).
LastUpdated: 2023-04-25 10:34:46Z
By B+R UnitTest Helper Version: 2.0.1.59
*/
#include "UnitTest.h"

UNITTEST_TESTSET_DECLARATION  Set_BrbUaDtStructToUaSrvDateTime;
UNITTEST_TESTSET_DECLARATION  Set_BrbUaSrvDateTimeToDtStruct;
UNITTEST_TESTSET_DECLARATION  Set_BrbUaGetSrvTimeText;
UNITTEST_TESTSET_DECLARATION  Set_BrbUaGetRandomTimeZone;

UNITTEST_TESTSET_FIXTURES(utTestSets)
{
	new_TestSet(Set_BrbUaDtStructToUaSrvDateTime),
	new_TestSet(Set_BrbUaSrvDateTimeToDtStruct),
	new_TestSet(Set_BrbUaGetSrvTimeText),
	new_TestSet(Set_BrbUaGetRandomTimeZone),
};
UNTITTEST_TESTSET_HANDLER();
```

#### Set_BrbUaDtStructToUaSrvDateTime.c - Test set
```c
#include <bur/plctypes.h>

#ifdef _DEFAULT_INCLUDES
#include <AsDefault.h>
#endif

#include "UnitTest.h"
#include "BrbAsserts.h"
#include <string.h>

// NOLINTBEGIN(readability-*, bugprone-easily-swappable-parameters, bugprone-branch-clone, clang-diagnostic-invalid-utf8, clang-diagnostic-invalid-source-encoding, clang-diagnostic-pointer-arith, clang-diagnostic-strict-prototypes, clang-diagnostic-bad-function-cast, clang-analyzer-security.insecureAPI.*, hicpp-uppercase-literal-suffix, cppcoreguidelines-*, performance-*)
_TEST BrbUaDtStructToUaSrvDateTime_NulPtr(void)
{
	uintOut = BrbUaDtStructToUaSrvDateTime(0, &dtStructIn, 123);
	TEST_ASSERT_EQUAL_INT(eBRB_ERR_NULL_POINTER, uintOut);

	uintOut = BrbUaDtStructToUaSrvDateTime(&srvDateTimeIn, 0, 123);
	TEST_ASSERT_EQUAL_INT(eBRB_ERR_NULL_POINTER, uintOut);

	// Finished
	TEST_DONE;
}

_TEST BrbUaDtStructToUaSrvDateTime_Convert(void)
{
	dtStructIn.year = 2023;
	dtStructIn.month = 01;
	dtStructIn.day = 02;
	dtStructIn.hour = 03;
	dtStructIn.minute = 04;
	dtStructIn.second = 05;
	dtStructIn.millisec = 006;
	dtStructIn.microsec = 007;
	uintOut = BrbUaDtStructToUaSrvDateTime(&srvDateTimeIn, &dtStructIn, 123);
	TEST_ASSERT_EQUAL_INT(eBRB_ERR_OK, uintOut);
	TEST_ASSERT_EQUAL_INT(1672628645, srvDateTimeIn.DateTime);
	TEST_ASSERT_EQUAL_INT(6007123, srvDateTimeIn.NanoSeconds);

	// Finished
	TEST_DONE;
}

// NOLINTEND(readability-*, bugprone-easily-swappable-parameters, bugprone-branch-clone, clang-diagnostic-invalid-utf8, clang-diagnostic-invalid-source-encoding, clang-diagnostic-pointer-arith, clang-diagnostic-strict-prototypes, clang-diagnostic-bad-function-cast, clang-analyzer-security.insecureAPI.*, hicpp-uppercase-literal-suffix, cppcoreguidelines-*, performance-*)

/*
B+R UnitTest: This is generated code.
Do not edit! Do not move!
Description: UnitTest Testprogramm infrastructure (TestSet).
LastUpdated: 2023-04-25 07:49:47Z
By B+R UnitTest Helper Version: 2.0.1.59
*/
UNITTEST_FIXTURES(fixtures)
{
	new_TestFixture("BrbUaDtStructToUaSrvDateTime_NulPtr", BrbUaDtStructToUaSrvDateTime_NulPtr),
	new_TestFixture("BrbUaDtStructToUaSrvDateTime_Convert", BrbUaDtStructToUaSrvDateTime_Convert),
};

UNITTEST_CALLER_COMPLETE_EXPLICIT(Set_BrbUaDtStructToUaSrvDateTime, "Set_BrbUaDtStructToUaSrvDateTime", 0, 0, fixtures, 0, 0, 0);
```

#### Set_BrbUaSrvDateTimeToDtStruct.c - Test set
```c
#include <bur/plctypes.h>

#ifdef _DEFAULT_INCLUDES
#include <AsDefault.h>
#endif

#include "UnitTest.h"
#include "BrbAsserts.h"
#include <string.h>

// NOLINTBEGIN(readability-*, bugprone-easily-swappable-parameters, bugprone-branch-clone, clang-diagnostic-invalid-utf8, clang-diagnostic-invalid-source-encoding, clang-diagnostic-pointer-arith, clang-diagnostic-strict-prototypes, clang-diagnostic-bad-function-cast, clang-analyzer-security.insecureAPI.*, hicpp-uppercase-literal-suffix, cppcoreguidelines-*, performance-*)
_TEST BrbUaSrvDateTimeToDtStruct_NulPtr(void)
{
	uintOut = BrbUaSrvDateTimeToDtStruct(0, &srvDateTimeIn);
	TEST_ASSERT_EQUAL_INT(eBRB_ERR_NULL_POINTER, uintOut);

	uintOut = BrbUaSrvDateTimeToDtStruct(&dtStructIn, 0);
	TEST_ASSERT_EQUAL_INT(eBRB_ERR_NULL_POINTER, uintOut);

	// Finished
	TEST_DONE;
}

_TEST BrbUaSrvDateTimeToDtStruct_Convert(void)
{
	srvDateTimeIn.DateTime = BrbSetDt(2023, 1, 2, 3, 4, 5);
	srvDateTimeIn.NanoSeconds = 6007123;
	uintOut = BrbUaSrvDateTimeToDtStruct(&dtStructIn, &srvDateTimeIn);
	TEST_ASSERT_EQUAL_INT(eBRB_ERR_OK, uintOut);
	BRB_ASSERT_EQUAL_DTSTRUCT(2023, 1, 2, eBRB_WD_MONDAY, 3, 4, 5, 6, 7, &dtStructIn);

	// Finished
	TEST_DONE;
}

// NOLINTEND(readability-*, bugprone-easily-swappable-parameters, bugprone-branch-clone, clang-diagnostic-invalid-utf8, clang-diagnostic-invalid-source-encoding, clang-diagnostic-pointer-arith, clang-diagnostic-strict-prototypes, clang-diagnostic-bad-function-cast, clang-analyzer-security.insecureAPI.*, hicpp-uppercase-literal-suffix, cppcoreguidelines-*, performance-*)

/*
B+R UnitTest: This is generated code.
Do not edit! Do not move!
Description: UnitTest Testprogramm infrastructure (TestSet).
LastUpdated: 2023-04-25 07:49:47Z
By B+R UnitTest Helper Version: 2.0.1.59
*/
UNITTEST_FIXTURES(fixtures)
{
	new_TestFixture("BrbUaSrvDateTimeToDtStruct_NulPtr", BrbUaSrvDateTimeToDtStruct_NulPtr),
	new_TestFixture("BrbUaSrvDateTimeToDtStruct_Convert", BrbUaSrvDateTimeToDtStruct_Convert),
};

UNITTEST_CALLER_COMPLETE_EXPLICIT(Set_BrbUaSrvDateTimeToDtStruct, "Set_BrbUaSrvDateTimeToDtStruct", 0, 0, fixtures, 0, 0, 0);
```

#### Set_BrbUaGetSrvTimeText.c - Test set
```c
#include <bur/plctypes.h>

#ifdef _DEFAULT_INCLUDES
#include <AsDefault.h>
#endif

#include "UnitTest.h"
#include "BrbAsserts.h"
#include <string.h>

// NOLINTBEGIN(readability-*, bugprone-easily-swappable-parameters, bugprone-branch-clone, clang-diagnostic-invalid-utf8, clang-diagnostic-invalid-source-encoding, clang-diagnostic-pointer-arith, clang-diagnostic-strict-prototypes, clang-diagnostic-bad-function-cast, clang-analyzer-security.insecureAPI.*, hicpp-uppercase-literal-suffix, cppcoreguidelines-*, performance-*)
_TEST BrbUaGetSrvTimeText_NulPtr(void)
{
	uintOut = BrbUaGetSrvTimeText(0, stringIn0, sizeof(stringIn0), 0, stringIn1);
	TEST_ASSERT_EQUAL_INT(eBRB_ERR_NULL_POINTER, uintOut);

	uintOut = BrbUaGetSrvTimeText(&srvDateTimeIn, 0, sizeof(stringIn0), 0, stringIn1);
	TEST_ASSERT_EQUAL_INT(eBRB_ERR_NULL_POINTER, uintOut);

	uintOut = BrbUaGetSrvTimeText(&srvDateTimeIn, stringIn0, 0, 0, stringIn1);
	TEST_ASSERT_EQUAL_INT(eBRB_ERR_INVALID_PARAMETER , uintOut);

	uintOut = BrbUaGetSrvTimeText(&srvDateTimeIn, stringIn0, sizeof(stringIn0), 0, 0);
	TEST_ASSERT_EQUAL_INT(eBRB_ERR_NULL_POINTER, uintOut);

	// Finished
	TEST_DONE;
}

_TEST BrbUaGetSrvTimeText_Get(void)
{
	srvDateTimeIn.DateTime = BrbSetDt(2023, 1, 2, 3, 4, 5);
	srvDateTimeIn.NanoSeconds = 6007823;
	strcpy(stringIn1, "yyyy-mm-dd hh:MM:ss:milms:micus:nanns");
	uintOut = BrbUaGetSrvTimeText(&srvDateTimeIn, stringIn0, sizeof(stringIn0), 0, stringIn1);
	TEST_ASSERT_EQUAL_INT(eBRB_ERR_OK, uintOut);
	TEST_ASSERT_EQUAL_STRING("2023-01-02 03:04:05:006ms:007us:823ns", stringIn0);

	srvDateTimeIn.DateTime = BrbSetDt(2023, 1, 2, 3, 4, 5);
	srvDateTimeIn.NanoSeconds = 6007823;
	strcpy(stringIn1, "yyyy-mm-dd hh:MM:ss:milms:micus:nanns");
	uintOut = BrbUaGetSrvTimeText(&srvDateTimeIn, stringIn0, sizeof(stringIn0), 60, stringIn1);
	TEST_ASSERT_EQUAL_INT(eBRB_ERR_OK, uintOut);
	TEST_ASSERT_EQUAL_STRING("2023-01-02 04:04:05:006ms:007us:823ns", stringIn0);

	// Finished
	TEST_DONE;
}

// NOLINTEND(readability-*, bugprone-easily-swappable-parameters, bugprone-branch-clone, clang-diagnostic-invalid-utf8, clang-diagnostic-invalid-source-encoding, clang-diagnostic-pointer-arith, clang-diagnostic-strict-prototypes, clang-diagnostic-bad-function-cast, clang-analyzer-security.insecureAPI.*, hicpp-uppercase-literal-suffix, cppcoreguidelines-*, performance-*)

/*
B+R UnitTest: This is generated code.
Do not edit! Do not move!
Description: UnitTest Testprogramm infrastructure (TestSet).
LastUpdated: 2023-04-25 07:55:27Z
By B+R UnitTest Helper Version: 2.0.1.59
*/
UNITTEST_FIXTURES(fixtures)
{
	new_TestFixture("BrbUaGetSrvTimeText_NulPtr", BrbUaGetSrvTimeText_NulPtr),
	new_TestFixture("BrbUaGetSrvTimeText_Get", BrbUaGetSrvTimeText_Get),
};

UNITTEST_CALLER_COMPLETE_EXPLICIT(Set_BrbUaGetSrvTimeText, "Set_BrbUaGetSrvTimeText", 0, 0, fixtures, 0, 0, 0);
```

#### Set_BrbUaGetRandomTimeZone.c - Test set
```c
#include <bur/plctypes.h>

#ifdef _DEFAULT_INCLUDES
#include <AsDefault.h>
#endif

#include "UnitTest.h"
#include "BrbAsserts.h"
#include <string.h>

// NOLINTBEGIN(readability-*, bugprone-easily-swappable-parameters, bugprone-branch-clone, clang-diagnostic-invalid-utf8, clang-diagnostic-invalid-source-encoding, clang-diagnostic-pointer-arith, clang-diagnostic-strict-prototypes, clang-diagnostic-bad-function-cast, clang-analyzer-security.insecureAPI.*, hicpp-uppercase-literal-suffix, cppcoreguidelines-*, performance-*)
_TEST BrbUaGetRandomTimeZone_NulPtr(void)
{
	dwordOut = BrbUaGetRandomTimeZone(0);
	TEST_ASSERT_EQUAL_INT(0x80460000, dwordOut); // = Bad_StructureMissing

	// Finished
	TEST_DONE;
}

_TEST BrbUaGetRandomTimeZone_Get(void)
{
	dwordOut = BrbUaGetRandomTimeZone(&timeZoneDataIn);
	TEST_ASSERT_EQUAL_INT(0x00000000, dwordOut);

	// Finished
	TEST_DONE;
}

// NOLINTEND(readability-*, bugprone-easily-swappable-parameters, bugprone-branch-clone, clang-diagnostic-invalid-utf8, clang-diagnostic-invalid-source-encoding, clang-diagnostic-pointer-arith, clang-diagnostic-strict-prototypes, clang-diagnostic-bad-function-cast, clang-analyzer-security.insecureAPI.*, hicpp-uppercase-literal-suffix, cppcoreguidelines-*, performance-*)

/*
B+R UnitTest: This is generated code.
Do not edit! Do not move!
Description: UnitTest Testprogramm infrastructure (TestSet).
LastUpdated: 2023-04-25 10:34:46Z
By B+R UnitTest Helper Version: 2.0.1.59
*/
UNITTEST_FIXTURES(fixtures)
{
	new_TestFixture("BrbUaGetRandomTimeZone_NulPtr", BrbUaGetRandomTimeZone_NulPtr),
	new_TestFixture("BrbUaGetRandomTimeZone_Get", BrbUaGetRandomTimeZone_Get),
};

UNITTEST_CALLER_COMPLETE_EXPLICIT(Set_BrbUaGetRandomTimeZone, "Set_BrbUaGetRandomTimeZone", 0, 0, fixtures, 0, 0, 0);
```

### Program Logical/UnitTests/UtBrbLibUa/UtBrbUaAdditional (ANSIC) - UnitTests

#### variables.var - Name the suite and add PVs for the program
```iecst
(********************************************************************
 * COPYRIGHT --
 ********************************************************************
 * Program: utTemplate_automated
 * File: variables.var
 * Author: -
 * Created: -
 ********************************************************************
 * Local variables of program utTemplate_automated
 ********************************************************************)
(*Describe the test*)
VAR
	Testsuite : UtMgrTestSuite := (Name:='BrbUaAdditional',Description:='(Optional field)Template for use with helper tool. Reference or add this program in the package "TS_UnitTest_UpdateTestPrograms"',Type:=utMgrTEST_TYPE_C,MetaInformation:='(Optional field):To be filled');
END_VAR
(*Input variables for testing*)
VAR
	guidStringIn : BrUaGuidString;
	xmlElementIn : BrUaXmlElement;
END_VAR
(*Functionblock instances for testing*)
(*Output variables for testing*)
VAR
	dwordOut : DWORD;
END_VAR
```

#### autoGeneratedFile.c - Auto generated code - list of all test sets in the program
```c
/*
B+R UnitTest: This is generated code.
Do not edit! Do not move!
Description: UnitTest Testprogramm infrastructure (List of TestSets).
LastUpdated: 2023-04-25 10:50:15Z
By B+R UnitTest Helper Version: 2.0.1.59
*/
#include "UnitTest.h"

UNITTEST_TESTSET_DECLARATION  Set_BrbUaGetRandomGuidString;
UNITTEST_TESTSET_DECLARATION  Set_BrbUaGetRandomXmlElement;

UNITTEST_TESTSET_FIXTURES(utTestSets)
{
	new_TestSet(Set_BrbUaGetRandomGuidString),
	new_TestSet(Set_BrbUaGetRandomXmlElement),
};
UNTITTEST_TESTSET_HANDLER();
```

#### Set_BrbUaGetRandomGuidString.c - Test set
```c
#include <bur/plctypes.h>

#ifdef _DEFAULT_INCLUDES
#include <AsDefault.h>
#endif

#include "UnitTest.h"
#include "BrbAsserts.h"
#include <string.h>

// NOLINTBEGIN(readability-*, bugprone-easily-swappable-parameters, bugprone-branch-clone, clang-diagnostic-invalid-utf8, clang-diagnostic-invalid-source-encoding, clang-diagnostic-pointer-arith, clang-diagnostic-strict-prototypes, clang-diagnostic-bad-function-cast, clang-analyzer-security.insecureAPI.*, hicpp-uppercase-literal-suffix, cppcoreguidelines-*, performance-*)
_TEST BrbUaGetRandomGuidString_NulPtr(void)
{
	dwordOut = BrbUaGetRandomGuidString(0, sizeof(guidStringIn), 1);
	TEST_ASSERT_EQUAL_INT(0x80460000, dwordOut); // = Bad_StructureMissing

	// Finished
	TEST_DONE;
}

_TEST BrbUaGetRandomGuidString_WithSep(void)
{
	dwordOut = BrbUaGetRandomGuidString(&guidStringIn, sizeof(guidStringIn), 1);
	TEST_ASSERT_EQUAL_INT(0x00000000, dwordOut); // = Good
	BRB_ASSERT_EQUAL_UDINT(36, strlen((STRING*)&guidStringIn));
	BRB_ASSERT_EQUAL_UDINT(4, BrbStringCountText(guidStringIn, "-", sizeof(guidStringIn)));
	TEST_ASSERT_EQUAL_INT('-', guidStringIn[8]);
	TEST_ASSERT_EQUAL_INT('-', guidStringIn[13]);
	TEST_ASSERT_EQUAL_INT('-', guidStringIn[18]);
	TEST_ASSERT_EQUAL_INT('-', guidStringIn[23]);

	// Finished
	TEST_DONE;
}

_TEST BrbUaGetRandomGuidString_WithoutSep(void)
{
	dwordOut = BrbUaGetRandomGuidString(&guidStringIn, sizeof(guidStringIn), 0);
	TEST_ASSERT_EQUAL_INT(0x00000000, dwordOut); // = Good
	BRB_ASSERT_EQUAL_UDINT(32, strlen((STRING*)&guidStringIn));
	BRB_ASSERT_EQUAL_UDINT(0, BrbStringCountText(guidStringIn, "-", sizeof(guidStringIn)));

	// Finished
	TEST_DONE;
}
// NOLINTEND(readability-*, bugprone-easily-swappable-parameters, bugprone-branch-clone, clang-diagnostic-invalid-utf8, clang-diagnostic-invalid-source-encoding, clang-diagnostic-pointer-arith, clang-diagnostic-strict-prototypes, clang-diagnostic-bad-function-cast, clang-analyzer-security.insecureAPI.*, hicpp-uppercase-literal-suffix, cppcoreguidelines-*, performance-*)

/*
B+R UnitTest: This is generated code.
Do not edit! Do not move!
Description: UnitTest Testprogramm infrastructure (TestSet).
LastUpdated: 2023-05-04 06:45:07Z
By B+R UnitTest Helper Version: 2.0.1.59
*/
UNITTEST_FIXTURES(fixtures)
{
	new_TestFixture("BrbUaGetRandomGuidString_NulPtr", BrbUaGetRandomGuidString_NulPtr),
	new_TestFixture("BrbUaGetRandomGuidString_WithSep", BrbUaGetRandomGuidString_WithSep),
	new_TestFixture("BrbUaGetRandomGuidString_WithoutSep", BrbUaGetRandomGuidString_WithoutSep),
};

UNITTEST_CALLER_COMPLETE_EXPLICIT(Set_BrbUaGetRandomGuidString, "Set_BrbUaGetRandomGuidString", 0, 0, fixtures, 0, 0, 0);
```

#### Set_BrbUaGetRandomXmlElement.c - Test set
```c
#include <bur/plctypes.h>

#ifdef _DEFAULT_INCLUDES
#include <AsDefault.h>
#endif

#include "UnitTest.h"
#include "BrbAsserts.h"
#include <string.h>

// NOLINTBEGIN(readability-*, bugprone-easily-swappable-parameters, bugprone-branch-clone, clang-diagnostic-invalid-utf8, clang-diagnostic-invalid-source-encoding, clang-diagnostic-pointer-arith, clang-diagnostic-strict-prototypes, clang-diagnostic-bad-function-cast, clang-analyzer-security.insecureAPI.*, hicpp-uppercase-literal-suffix, cppcoreguidelines-*, performance-*)
_TEST BrbUaGetRandomXmlElement_NulPtr(void)
{
	dwordOut = BrbUaGetRandomXmlElement(0);
	TEST_ASSERT_EQUAL_INT(0x80460000, dwordOut); // = Bad_StructureMissing

	// Finished
	TEST_DONE;
}

_TEST BrbUaGetRandomXmlElement_Status(void)
{
	dwordOut = BrbUaGetRandomXmlElement(&xmlElementIn);
	TEST_ASSERT_EQUAL_INT(0x00000000, dwordOut); // = Good

	// Finished
	TEST_DONE;
}

// NOLINTEND(readability-*, bugprone-easily-swappable-parameters, bugprone-branch-clone, clang-diagnostic-invalid-utf8, clang-diagnostic-invalid-source-encoding, clang-diagnostic-pointer-arith, clang-diagnostic-strict-prototypes, clang-diagnostic-bad-function-cast, clang-analyzer-security.insecureAPI.*, hicpp-uppercase-literal-suffix, cppcoreguidelines-*, performance-*)

/*
B+R UnitTest: This is generated code.
Do not edit! Do not move!
Description: UnitTest Testprogramm infrastructure (TestSet).
LastUpdated: 2023-04-25 10:50:15Z
By B+R UnitTest Helper Version: 2.0.1.59
*/
UNITTEST_FIXTURES(fixtures)
{
	new_TestFixture("BrbUaGetRandomXmlElement_NulPtr", BrbUaGetRandomXmlElement_NulPtr),
	new_TestFixture("BrbUaGetRandomXmlElement_Status", BrbUaGetRandomXmlElement_Status),
};

UNITTEST_CALLER_COMPLETE_EXPLICIT(Set_BrbUaGetRandomXmlElement, "Set_BrbUaGetRandomXmlElement", 0, 0, fixtures, 0, 0, 0);
```

### Program Logical/UnitTests/UtBrbLibUa/UtBrbUaClient (ANSIC) - UnitTests

#### variables.var - Name the suite and add PVs for the program
```iecst
(********************************************************************
 * COPYRIGHT --
 ********************************************************************
 * Program: utTemplate_automated
 * File: variables.var
 * Author: -
 * Created: -
 ********************************************************************
 * Local variables of program utTemplate_automated
 ********************************************************************)
(*Describe the test*)
VAR
	Testsuite : UtMgrTestSuite := (Name:='BrbUaClient',Description:='(Optional field)Template for use with helper tool. Reference or add this program in the package "TS_UnitTest_UpdateTestPrograms"',Type:=utMgrTEST_TYPE_C,MetaInformation:='(Optional field):To be filled');
END_VAR
(*Input variables for testing*)
VAR
	connectionStatus : UAConnectionStatus;
	stringIn0 : STRING[64];
END_VAR
(*Functionblock instances for testing*)
(*Output variables for testing*)
VAR
	dwordOut : DWORD;
END_VAR
```

#### autoGeneratedFile.c - Auto generated code - list of all test sets in the program
```c
/*
B+R UnitTest: This is generated code.
Do not edit! Do not move!
Description: UnitTest Testprogramm infrastructure (List of TestSets).
LastUpdated: 2023-04-25 10:54:48Z
By B+R UnitTest Helper Version: 2.0.1.59
*/
#include "UnitTest.h"

UNITTEST_TESTSET_DECLARATION  Set_BrbUaGetConnectionStatusText;

UNITTEST_TESTSET_FIXTURES(utTestSets)
{
	new_TestSet(Set_BrbUaGetConnectionStatusText),
};
UNTITTEST_TESTSET_HANDLER();
```

#### Set_BrbUaGetConnectionStatusText.c - Test set
```c
#include <bur/plctypes.h>

#ifdef _DEFAULT_INCLUDES
#include <AsDefault.h>
#endif

#include "UnitTest.h"
#include "BrbAsserts.h"
#include <string.h>

// NOLINTBEGIN(readability-*, bugprone-easily-swappable-parameters, bugprone-branch-clone, clang-diagnostic-invalid-utf8, clang-diagnostic-invalid-source-encoding, clang-diagnostic-pointer-arith, clang-diagnostic-strict-prototypes, clang-diagnostic-bad-function-cast, clang-analyzer-security.insecureAPI.*, hicpp-uppercase-literal-suffix, cppcoreguidelines-*, performance-*)
_TEST BrbUaGetConnectionStatusText_NulPtr(void)
{
	dwordOut = BrbUaGetConnectionStatusText(0, 0, 0);
	TEST_ASSERT_EQUAL_INT(0x80460000, dwordOut); // = Bad_StructureMissing

	// Finished
	TEST_DONE;
}

_TEST BrbUaGetConnectionStatusText_Get(void)
{
	connectionStatus = UACS_Connected;
	dwordOut = BrbUaGetConnectionStatusText(connectionStatus, stringIn0, sizeof(stringIn0));
	TEST_ASSERT_EQUAL_INT(0x00000000, dwordOut); // = Good
	TEST_ASSERT_EQUAL_STRING("Connected", stringIn0);

	// Finished
	TEST_DONE;
}

// NOLINTEND(readability-*, bugprone-easily-swappable-parameters, bugprone-branch-clone, clang-diagnostic-invalid-utf8, clang-diagnostic-invalid-source-encoding, clang-diagnostic-pointer-arith, clang-diagnostic-strict-prototypes, clang-diagnostic-bad-function-cast, clang-analyzer-security.insecureAPI.*, hicpp-uppercase-literal-suffix, cppcoreguidelines-*, performance-*)

/*
B+R UnitTest: This is generated code.
Do not edit! Do not move!
Description: UnitTest Testprogramm infrastructure (TestSet).
LastUpdated: 2023-04-25 10:54:48Z
By B+R UnitTest Helper Version: 2.0.1.59
*/
UNITTEST_FIXTURES(fixtures)
{
	new_TestFixture("BrbUaGetConnectionStatusText_NulPtr", BrbUaGetConnectionStatusText_NulPtr),
	new_TestFixture("BrbUaGetConnectionStatusText_Get", BrbUaGetConnectionStatusText_Get),
};

UNITTEST_CALLER_COMPLETE_EXPLICIT(Set_BrbUaGetConnectionStatusText, "Set_BrbUaGetConnectionStatusText", 0, 0, fixtures, 0, 0, 0);
```

### Program Logical/UnitTests/UtBrbLibUa/UtBrbUaServer (ANSIC) - UnitTests

#### variables.var - Name the suite and add PVs for the program
```iecst
(********************************************************************
 * COPYRIGHT --
 ********************************************************************
 * Program: utTemplate_automated
 * File: variables.var
 * Author: -
 * Created: -
 ********************************************************************
 * Local variables of program utTemplate_automated
 ********************************************************************)
(*Describe the test*)
VAR
	Testsuite : UtMgrTestSuite := (Name:='BrbUaServer',Description:='(Optional field)Template for use with helper tool. Reference or add this program in the package "TS_UnitTest_UpdateTestPrograms"',Type:=utMgrTEST_TYPE_C,MetaInformation:='(Optional field):To be filled');
END_VAR
(*Input variables for testing*)
VAR
	methodOperationAction : UaMethodOperateAction;
	stringIn0 : STRING[64];
END_VAR
(*Functionblock instances for testing*)
(*Output variables for testing*)
VAR
	dwordOut : DWORD;
END_VAR
```

#### autoGeneratedFile.c - Auto generated code - list of all test sets in the program
```c
/*
B+R UnitTest: This is generated code.
Do not edit! Do not move!
Description: UnitTest Testprogramm infrastructure (List of TestSets).
LastUpdated: 2023-04-25 13:44:36Z
By B+R UnitTest Helper Version: 2.0.1.59
*/
#include "UnitTest.h"

UNITTEST_TESTSET_DECLARATION  Set_BrbUaSrvGetMethodOperateText;

UNITTEST_TESTSET_FIXTURES(utTestSets)
{
	new_TestSet(Set_BrbUaSrvGetMethodOperateText),
};
UNTITTEST_TESTSET_HANDLER();
```
